(* Logix 5000 project; controller cow Emulate 5570 rev 36.11; software revision 36.00; part 3 of 6 *)

VAR_GLOBAL   (* controller tags *)
   B111 : MotorX := (InterLock := 1, SP := 1, LSK := 1);
   B113 : MotorX := (LSK := 1);
   B116 : MotorX := (LSK := 1);
   B126 : MotorX := (InterLock := 1, SP := 1, LSK := 1, CLEAN := 1);
   B160 : MotorX := (LSK := 1);
   B280 : Divider := (LS3 := 1, LS_ON := 1, Simulate := 3);
   B3 : INT[50] := ([0] := 1, [2] := 896, [3] := 15824, [6] := 24508, [7] := 19455, [8] := 677, [16] := 7, [18] := 1503, [22] := 4736, [23] := 160, [24] := 2145, [26] := -22782, [28] := -22484, [29] := 21, [30] := 768, [33] := 11328, [34] := 24701, [35] := 12288, [40] := 4, [41] := 4, [42] := 816, [43] := -19680, [44] := -21846, [45] := -32054, [46] := 194, [47] := 26775);
   B353 : Gate := (LSK := 1);
   B354 : Gate := (LSK := 1);
   B361 : Branch_SV2 := (LSX := 1, GLX := 1);
   B362 : Branch_SV2 := (LSY := 1, GLY := 1);
   B363 : Branch_SV2 := (LSY := 1, GLY := 1);
   B364 : Branch_SV2 := (LSY := 1, GLY := 1);
   B365 : Branch_SV2 := (LSX := 1, GLX := 1);
   B367 : Branch_SV2 := (LSX := 1, GLX := 1);
   B410 : MotorX := (LSK := 1);
   B420 : MotorX := (LSK := 1);
   Bin01 : ALIAS FOR rcp_Big_Bin[0];
   Bin02 : ALIAS FOR rcp_Big_Bin[1];
   Bin03 : ALIAS FOR rcp_Big_Bin[2];
   Bin04 : ALIAS FOR rcp_Big_Bin[3];
   Bin05 : ALIAS FOR rcp_Big_Bin[4];
   Bin06 : ALIAS FOR rcp_Big_Bin[5];
   Bin07 : ALIAS FOR rcp_Big_Bin[6];
   Bin08 : ALIAS FOR rcp_Big_Bin[7];
   Bin09 : ALIAS FOR rcp_Big_Bin[8];
   Bin10 : ALIAS FOR rcp_Big_Bin[9];
   Bin11 : ALIAS FOR rcp_Big_Bin[10];
   Bin12 : ALIAS FOR rcp_Big_Bin[11];
   Bin13 : ALIAS FOR rcp_Big_Bin[12];
   Bin14 : ALIAS FOR rcp_Big_Bin[13];
   Bin15 : ALIAS FOR rcp_Big_Bin[14];
   Bin16 : ALIAS FOR rcp_Big_Bin[15];
   Buf_LenSent : DINT := 8;
   D121 : MotorX := (LSK := 1);
   D162 : MotorX := (LSK := 1);
   D163 : MotorX := (LSK := 1);
   D164 : MotorX := (LSK := 1);
   D230 : MotorX := (LSK := 1);
   D361 : Branch_SV2 := (LSY := 1, GLY := 1);
   D380 : MotorX := (LSK := 1);
   D411 : MotorX := (LSK := 1);
   D421 : MotorX := (LSK := 1);
   DateTimes : STRING := '2026/06/05  08:19:56';
   Delete_All_MSG : MESSAGE;
        MessageParameters(ServiceCode := 16#0051, ...)
   E112 : MotorX := (LL := 1, Auto := 1, LSK := 1);   // B112
   E112_Have : BOOL;
   E112_Have_Flash : BOOL;
   E120 : MotorX := (Auto := 1, SP := 1, LSK := 1, CLEAN := 1);   // B120
   E141 : MotorX := (Auto := 1, SP := 1, LSK := 1);   // B141
   E142 : MotorX := (Auto := 1, SP := 1, LSK := 1);
   E143 : MotorX := (Auto := 1, LSK := 1);
   E144 : MotorX := (Auto := 1, LSK := 1);
   E145 : MotorX := (Auto := 1, SP := 1, LSK := 1);
   E146 : MotorX := (Auto := 1, LSK := 1);
   E147 : MotorX := (Auto := 1, LSK := 1);
   E148 : MotorX := (Auto := 1, LSK := 1);
   E149 : MotorX := (Auto := 1, LSK := 1);
   E14A : MotorX := (Auto := 1, LSK := 1);
   E14B : MotorX := (Auto := 1, LSK := 1);
   E14C : MotorX := (Auto := 1, LSK := 1);
   E14D : MotorX := (Auto := 1, LSK := 1);
   E14E : MotorX := (Auto := 1, LSK := 1);
   E14F : MotorX := (Auto := 1, LSK := 1);
   E14G : MotorX := (Auto := 1, LSK := 1);
   E331 : SCALE_WEIGHT;
   E340 : Valve := (LSK := 1, Auto := 1, PB := 1);
   E351 : Valve := (LSK := 1, Auto := 1);
   E352 : Valve := (LSK := 1, Auto := 1);
   E45A : Air_Hammer := (MotorType := 1);
   E45B : Air_Hammer;
   E45C : Air_Hammer;
   EINV : Inverter := (Manual_HZ := 10);
   F090 : MotorX := (LSK := 1);
   F124 : MotorX := (LSK := 1);
   F125 : MotorX := (LSK := 1);
   F140 : MotorX := (LSK := 1);
   F167 : MotorX := (LSK := 1);
   F168 : MotorX := (LSK := 1);
   F240 : MotorX := (LSK := 1);
   F270 : MotorX := (LSK := 1);
   F363 : Branch_SV2 := (LSY := 1, GLY := 1);
   F364 : Branch_SV2 := (LSY := 1, GLY := 1);
   F413 : MotorX := (LSK := 1);
   F441 : MotorX := (LSK := 1);
   F560 : MotorX := (LSK := 1);
   F561 : MotorX := (LSK := 1);
   LED0_Create_Sock_MSG : MESSAGE;
        MessageParameters(ServiceCode := 16#004b, LocalElement := LED_SOCKET[0], DestinationTag := LED_Instance[0], ...)
   LED0_Write_Data_MSG : MESSAGE;
        MessageParameters(ServiceCode := 16#004e, LocalElement := LED_Write_Data_Out[0], DestinationTag := Buf_LenSent, ...)
   LED_Batch_seq : DINT := 1;
   LED_Batch_Total : ALIAS FOR rcp_Recipe.BatchSet;
   Led_Hand_PartNumber : DINT;
   Led_Hand_RealWeight : REAL;
   LED_Hand_SetWeight : REAL;
   LED_Instance : DINT[16] := ([0] := 18562, [1] := 31683, [2] := 27332, [3] := 24000, [4] := 22593, [5] := 19589, [6] := 24710, [7] := 29255, [8] := 16968);
   LED_SOCKET : REQUEST_PARAMETERS[16] := ([0].Type := 2, [0].Addr.Family := 2, [0].Addr.Port := 123, [1].Type := 2, [1].Addr.Family := 2, [1].Addr.Port := 121, [2].Type := 2, [2].Addr.Family := 2, [2].Addr.Port := 221, [3].Type := 2, [3].Addr.Family := 2, [3].Addr.Port := 122, [4].Type := 2, [4].Addr.Family := 2, [4].Addr.Port := 222, [5].Type := 2, [5].Addr.Family := 2, [5].Addr.Port := 223, [6].Type := 2, [6].Addr.Family := 2, [6].Addr.Port := 124, [7].Type := 2, [7].Addr.Family := 2, [7].Addr.Port := 125, [8].Type := 2, [8].Addr.Family := 2, [8].Addr.Port := 226);
   Led_string : STRING[16] := ([0] := 'Test$00$00$00$00$00$00 2-1      ', [1] := '2026/04/29  10:28:13', [2] := '730000600  100.0 Kg ', [3] := 'BIN:41 3016E 5.00 t ', [4] := 'BIN:34 2410$00$00- 6.00t', [5] := '2026/04/29  10:28:13', [6] := 'S19-B8-2001B$00-99.0t ', [7] := 'S0-B139-3015$00$00- 3.0t', [8] := 'BIN1 2001F$00-30.00t  ');
   LED_Write_Data_Out : WRT_DATA[16] := ([0].Timeout := 20000, [0].ToAddr.Family := 2, [0].ToAddr.Port := 8001, [0].ToAddr.Addr := 16#c101_017b, [0].Buffer.LEN := 31, [0].Buffer.BUFF[0] := 2, [0].Buffer.BUFF[1] := 90, [0].Buffer.BUFF[2] := 48, [0].Buffer.BUFF[3] := -95, [0].Buffer.BUFF[4] := 1, [0].Buffer.BUFF[5] := 1, [0].Buffer.BUFF[6] := 78, [0].Buffer.BUFF[7] := -48, [0].Buffer.BUFF[8] := 55, [0].Buffer.BUFF[9] := 55, [0].Buffer.BUFF[10] := 48, [0].Buffer.BUFF[11] := 48, [0].Buffer.BUFF[12] := 51, [0].Buffer.BUFF[13] := 49, [0].Buffer.BUFF[14] := 51, [0].Buffer.BUFF[15] := 57, [0].Buffer.BUFF[16] := 48, [0].Buffer.BUFF[17] := 100, [0].Buffer.BUFF[18] := 32, [0].Buffer.BUFF[19] := 53, [0].Buffer.BUFF[20] := 45, [0].Buffer.BUFF[21] := 51, [0].Buffer.BUFF[22] := 32, [0].Buffer.BUFF[23] := 32, [0].Buffer.BUFF[24] := 32, [0].Buffer.BUFF[25] := 32, [0].Buffer.BUFF[26] := 32, [0].Buffer.BUFF[27] := 32, [0].Buffer.BUFF[28] := 82, [0].Buffer.BUFF[29] := 80, [0].Buffer.BUFF[30] := 3, [0].Buffer.BUFF[31] := 46, [0].Buffer.BUFF[32] := 48, [0].Buffer.BUFF[33] := 82, [0].Buffer.BUFF[34] := 51, [0].Buffer.BUFF[35] := 3, [0].Buffer.BUFF[84] := 31, [0].Buffer.BUFF[88] := 2, [0].Buffer.BUFF[89] := 90, [0].Buffer.BUFF[90] := 48, [0].Buffer.BUFF[91] := -95, [0].Buffer.BUFF[92] := 1, [0].Buffer.BUFF[93] := 1, [0].Buffer.BUFF[94] := 78, [0].Buffer.BUFF[95] := -48, [0].Buffer.BUFF[96] := 50, [0].Buffer.BUFF[97] := 48, [0].Buffer.BUFF[98] := 50, [0].Buffer.BUFF[99] := 54, [0].Buffer.BUFF[100] := 47, [0].Buffer.BUFF[101] := 48, [0].Buffer.BUFF[102] := 52, [0].Buffer.BUFF[103] := 47, [0].Buffer.BUFF[104] := 50, [0].Buffer.BUFF[105] := 57,
        [0].Buffer.BUFF[106] := 32, [0].Buffer.BUFF[107] := 32, [0].Buffer.BUFF[108] := 49, [0].Buffer.BUFF[109] := 48, [0].Buffer.BUFF[110] := 58, [0].Buffer.BUFF[111] := 50, [0].Buffer.BUFF[112] := 56, [0].Buffer.BUFF[113] := 58, [0].Buffer.BUFF[114] := 48, [0].Buffer.BUFF[115] := 56, [0].Buffer.BUFF[116] := 82, [0].Buffer.BUFF[117] := 13, [0].Buffer.BUFF[118] := 3, [0].Buffer.BUFF[172] := 31, [0].Buffer.BUFF[176] := 2, [0].Buffer.BUFF[177] := 90, [0].Buffer.BUFF[178] := 48, [0].Buffer.BUFF[179] := -95, [0].Buffer.BUFF[180] := 1, [0].Buffer.BUFF[181] := 1, [0].Buffer.BUFF[182] := 78, [0].Buffer.BUFF[183] := -48, [0].Buffer.BUFF[184] := 55, [0].Buffer.BUFF[185] := 51, [0].Buffer.BUFF[186] := 48, [0].Buffer.BUFF[187] := 48, [0].Buffer.BUFF[188] := 48, [0].Buffer.BUFF[189] := 48, [0].Buffer.BUFF[190] := 54, [0].Buffer.BUFF[191] := 48, [0].Buffer.BUFF[192] := 48, [0].Buffer.BUFF[193] := 32, [0].Buffer.BUFF[194] := 32, [0].Buffer.BUFF[195] := 49, [0].Buffer.BUFF[196] := 48, [0].Buffer.BUFF[197] := 48, [0].Buffer.BUFF[198] := 46, [0].Buffer.BUFF[199] := 48, [0].Buffer.BUFF[200] := 32, [0].Buffer.BUFF[201] := 75, [0].Buffer.BUFF[202] := 103, [0].Buffer.BUFF[203] := 32, [0].Buffer.BUFF[204] := 82, [0].Buffer.BUFF[205] := 54, [0].Buffer.BUFF[206] := 3, [0].Buffer.BUFF[260] := 31, [0].Buffer.BUFF[264] := 2, [0].Buffer.BUFF[265] := 90, [0].Buffer.BUFF[266] := 48, [0].Buffer.BUFF[267] := -95, [0].Buffer.BUFF[268] := 1, [0].Buffer.BUFF[269] := 1, [0].Buffer.BUFF[270] := 78, [0].Buffer.BUFF[271] := -48, [0].Buffer.BUFF[272] := 66, [0].Buffer.BUFF[273] := 73, [0].Buffer.BUFF[274] := 78, [0].Buffer.BUFF[275] := 58, [0].Buffer.BUFF[276] := 52, [0].Buffer.BUFF[277] := 49,
        [0].Buffer.BUFF[278] := 32, [0].Buffer.BUFF[279] := 51, [0].Buffer.BUFF[280] := 48, [0].Buffer.BUFF[281] := 49, [0].Buffer.BUFF[282] := 54, [0].Buffer.BUFF[283] := 69, [0].Buffer.BUFF[284] := 32, [0].Buffer.BUFF[285] := 53, [0].Buffer.BUFF[286] := 46, [0].Buffer.BUFF[287] := 48, [0].Buffer.BUFF[288] := 48, [0].Buffer.BUFF[289] := 32, [0].Buffer.BUFF[290] := 116, [0].Buffer.BUFF[291] := 32, [0].Buffer.BUFF[292] := 82, [0].Buffer.BUFF[293] := 83, [0].Buffer.BUFF[294] := 3, [0].Buffer.BUFF[348] := 31, [0].Buffer.BUFF[352] := 2, [0].Buffer.BUFF[353] := 90, [0].Buffer.BUFF[354] := 48, [0].Buffer.BUFF[355] := -95, [0].Buffer.BUFF[356] := 1, [0].Buffer.BUFF[357] := 1, [0].Buffer.BUFF[358] := 78, [0].Buffer.BUFF[359] := -48, [0].Buffer.BUFF[360] := 66, [0].Buffer.BUFF[361] := 73, [0].Buffer.BUFF[362] := 78, [0].Buffer.BUFF[363] := 58, [0].Buffer.BUFF[364] := 51, [0].Buffer.BUFF[365] := 52, [0].Buffer.BUFF[366] := 32, [0].Buffer.BUFF[367] := 50, [0].Buffer.BUFF[368] := 52, [0].Buffer.BUFF[369] := 49, [0].Buffer.BUFF[370] := 48, [0].Buffer.BUFF[373] := 45, [0].Buffer.BUFF[374] := 32, [0].Buffer.BUFF[375] := 54, [0].Buffer.BUFF[376] := 46, [0].Buffer.BUFF[377] := 48, [0].Buffer.BUFF[378] := 48, [0].Buffer.BUFF[379] := 116, [0].Buffer.BUFF[380] := 82, [0].Buffer.BUFF[381] := 57, [0].Buffer.BUFF[382] := 3, [0].Buffer.BUFF[436] := 31, [0].Buffer.BUFF[440] := 2, [0].Buffer.BUFF[441] := 90, [0].Buffer.BUFF[442] := 48, [0].Buffer.BUFF[443] := -95, [0].Buffer.BUFF[444] := 1, [0].Buffer.BUFF[445] := 1, [0].Buffer.BUFF[446] := 78, [0].Buffer.BUFF[447] := -48, [0].Buffer.BUFF[448] := 50, [0].Buffer.BUFF[449] := 48, [0].Buffer.BUFF[450] := 50, [0].Buffer.BUFF[451] := 54,
        [0].Buffer.BUFF[452] := 47, [0].Buffer.BUFF[453] := 48, [0].Buffer.BUFF[454] := 52, [0].Buffer.BUFF[455] := 47, [0].Buffer.BUFF[456] := 50, [0].Buffer.BUFF[457] := 57, [0].Buffer.BUFF[458] := 32, [0].Buffer.BUFF[459] := 32, [0].Buffer.BUFF[460] := 49, [0].Buffer.BUFF[461] := 48, [0].Buffer.BUFF[462] := 58, [0].Buffer.BUFF[463] := 50, [0].Buffer.BUFF[464] := 56, [0].Buffer.BUFF[465] := 58, [0].Buffer.BUFF[466] := 48, [0].Buffer.BUFF[467] := 56, [0].Buffer.BUFF[468] := 82, [0].Buffer.BUFF[469] := 13, [0].Buffer.BUFF[470] := 3, [1].ToAddr.Family := 2, [1].ToAddr.Port := 8001, [1].ToAddr.Addr := 16#c101_0179, [1].Buffer.LEN := 31, [1].Buffer.BUFF[0] := 2, [1].Buffer.BUFF[1] := 90, [1].Buffer.BUFF[2] := 48, [1].Buffer.BUFF[3] := -95, [1].Buffer.BUFF[4] := 1, [1].Buffer.BUFF[5] := 1, [1].Buffer.BUFF[6] := 78, [1].Buffer.BUFF[7] := -48, [1].Buffer.BUFF[8] := 50, [1].Buffer.BUFF[9] := 48, [1].Buffer.BUFF[10] := 50, [1].Buffer.BUFF[11] := 54, [1].Buffer.BUFF[12] := 47, [1].Buffer.BUFF[13] := 48, [1].Buffer.BUFF[14] := 52, [1].Buffer.BUFF[15] := 47, [1].Buffer.BUFF[16] := 50, [1].Buffer.BUFF[17] := 57, [1].Buffer.BUFF[18] := 32, [1].Buffer.BUFF[19] := 32, [1].Buffer.BUFF[20] := 49, [1].Buffer.BUFF[21] := 48, [1].Buffer.BUFF[22] := 58, [1].Buffer.BUFF[23] := 50, [1].Buffer.BUFF[24] := 56, [1].Buffer.BUFF[25] := 58, [1].Buffer.BUFF[26] := 48, [1].Buffer.BUFF[27] := 55, [1].Buffer.BUFF[28] := 82, [1].Buffer.BUFF[29] := 2, [1].Buffer.BUFF[30] := 3, [1].Buffer.BUFF[84] := 31, [1].Buffer.BUFF[88] := 2, [1].Buffer.BUFF[89] := 90, [1].Buffer.BUFF[90] := 48, [1].Buffer.BUFF[91] := -95, [1].Buffer.BUFF[92] := 1,
        [1].Buffer.BUFF[93] := 1, [1].Buffer.BUFF[94] := 78, [1].Buffer.BUFF[95] := -48, [1].Buffer.BUFF[96] := 55, [1].Buffer.BUFF[97] := 51, [1].Buffer.BUFF[98] := 48, [1].Buffer.BUFF[99] := 48, [1].Buffer.BUFF[100] := 48, [1].Buffer.BUFF[101] := 48, [1].Buffer.BUFF[102] := 54, [1].Buffer.BUFF[103] := 48, [1].Buffer.BUFF[104] := 48, [1].Buffer.BUFF[105] := 32, [1].Buffer.BUFF[106] := 32, [1].Buffer.BUFF[107] := 49, [1].Buffer.BUFF[108] := 48, [1].Buffer.BUFF[109] := 48, [1].Buffer.BUFF[110] := 46, [1].Buffer.BUFF[111] := 48, [1].Buffer.BUFF[112] := 32, [1].Buffer.BUFF[113] := 75, [1].Buffer.BUFF[114] := 103, [1].Buffer.BUFF[115] := 32, [1].Buffer.BUFF[116] := 82, [1].Buffer.BUFF[117] := 54, [1].Buffer.BUFF[118] := 3, [1].Buffer.BUFF[172] := 31, [1].Buffer.BUFF[176] := 2, [1].Buffer.BUFF[177] := 90, [1].Buffer.BUFF[178] := 48, [1].Buffer.BUFF[179] := -95, [1].Buffer.BUFF[180] := 1, [1].Buffer.BUFF[181] := 1, [1].Buffer.BUFF[182] := 78, [1].Buffer.BUFF[183] := -48, [1].Buffer.BUFF[184] := 66, [1].Buffer.BUFF[185] := 73, [1].Buffer.BUFF[186] := 78, [1].Buffer.BUFF[187] := 58, [1].Buffer.BUFF[188] := 52, [1].Buffer.BUFF[189] := 49, [1].Buffer.BUFF[190] := 32, [1].Buffer.BUFF[191] := 51, [1].Buffer.BUFF[192] := 48, [1].Buffer.BUFF[193] := 49, [1].Buffer.BUFF[194] := 54, [1].Buffer.BUFF[195] := 69, [1].Buffer.BUFF[196] := 32, [1].Buffer.BUFF[197] := 53, [1].Buffer.BUFF[198] := 46, [1].Buffer.BUFF[199] := 48, [1].Buffer.BUFF[200] := 48, [1].Buffer.BUFF[201] := 32, [1].Buffer.BUFF[202] := 116, [1].Buffer.BUFF[203] := 32, [1].Buffer.BUFF[204] := 82, [1].Buffer.BUFF[205] := 83, [1].Buffer.BUFF[206] := 3, [1].Buffer.BUFF[260] := 31, [1].Buffer.BUFF[264] := 2,
        [1].Buffer.BUFF[265] := 90, [1].Buffer.BUFF[266] := 48, [1].Buffer.BUFF[267] := -95, [1].Buffer.BUFF[268] := 1, [1].Buffer.BUFF[269] := 1, [1].Buffer.BUFF[270] := 78, [1].Buffer.BUFF[271] := -48, [1].Buffer.BUFF[272] := 66, [1].Buffer.BUFF[273] := 73, [1].Buffer.BUFF[274] := 78, [1].Buffer.BUFF[275] := 58, [1].Buffer.BUFF[276] := 51, [1].Buffer.BUFF[277] := 52, [1].Buffer.BUFF[278] := 32, [1].Buffer.BUFF[279] := 50, [1].Buffer.BUFF[280] := 52, [1].Buffer.BUFF[281] := 49, [1].Buffer.BUFF[282] := 48, [1].Buffer.BUFF[285] := 45, [1].Buffer.BUFF[286] := 32, [1].Buffer.BUFF[287] := 54, [1].Buffer.BUFF[288] := 46, [1].Buffer.BUFF[289] := 48, [1].Buffer.BUFF[290] := 48, [1].Buffer.BUFF[291] := 116, [1].Buffer.BUFF[292] := 82, [1].Buffer.BUFF[293] := 57, [1].Buffer.BUFF[294] := 3, [1].Buffer.BUFF[348] := 31, [1].Buffer.BUFF[352] := 2, [1].Buffer.BUFF[353] := 90, [1].Buffer.BUFF[354] := 48, [1].Buffer.BUFF[355] := -95, [1].Buffer.BUFF[356] := 1, [1].Buffer.BUFF[357] := 1, [1].Buffer.BUFF[358] := 78, [1].Buffer.BUFF[359] := -48, [1].Buffer.BUFF[360] := 50, [1].Buffer.BUFF[361] := 48, [1].Buffer.BUFF[362] := 50, [1].Buffer.BUFF[363] := 54, [1].Buffer.BUFF[364] := 47, [1].Buffer.BUFF[365] := 48, [1].Buffer.BUFF[366] := 52, [1].Buffer.BUFF[367] := 47, [1].Buffer.BUFF[368] := 50, [1].Buffer.BUFF[369] := 57, [1].Buffer.BUFF[370] := 32, [1].Buffer.BUFF[371] := 32, [1].Buffer.BUFF[372] := 49, [1].Buffer.BUFF[373] := 48, [1].Buffer.BUFF[374] := 58, [1].Buffer.BUFF[375] := 50, [1].Buffer.BUFF[376] := 56, [1].Buffer.BUFF[377] := 58, [1].Buffer.BUFF[378] := 48, [1].Buffer.BUFF[379] := 55, [1].Buffer.BUFF[380] := 82, [1].Buffer.BUFF[381] := 2, [1].Buffer.BUFF[382] := 3,
        [1].Buffer.BUFF[436] := 31, [1].Buffer.BUFF[440] := 2, [1].Buffer.BUFF[441] := 90, [1].Buffer.BUFF[442] := 48, [1].Buffer.BUFF[443] := -95, [1].Buffer.BUFF[444] := 1, [1].Buffer.BUFF[445] := 1, [1].Buffer.BUFF[446] := 78, [1].Buffer.BUFF[447] := -48, [1].Buffer.BUFF[448] := 83, [1].Buffer.BUFF[449] := 49, [1].Buffer.BUFF[450] := 57, [1].Buffer.BUFF[451] := 45, [1].Buffer.BUFF[452] := 66, [1].Buffer.BUFF[453] := 56, [1].Buffer.BUFF[454] := 45, [1].Buffer.BUFF[455] := 50, [1].Buffer.BUFF[456] := 48, [1].Buffer.BUFF[457] := 48, [1].Buffer.BUFF[458] := 49, [1].Buffer.BUFF[459] := 66, [1].Buffer.BUFF[461] := 45, [1].Buffer.BUFF[462] := 57, [1].Buffer.BUFF[463] := 57, [1].Buffer.BUFF[464] := 46, [1].Buffer.BUFF[465] := 48, [1].Buffer.BUFF[466] := 116, [1].Buffer.BUFF[467] := 32, [1].Buffer.BUFF[468] := 82, [1].Buffer.BUFF[470] := 3, [2].ToAddr.Family := 2, [2].ToAddr.Port := 8002, [2].ToAddr.Addr := 16#c101_0179, [2].Buffer.LEN := 31, [2].Buffer.BUFF[0] := 2, [2].Buffer.BUFF[1] := 90, [2].Buffer.BUFF[2] := 48, [2].Buffer.BUFF[3] := -95, [2].Buffer.BUFF[4] := 1, [2].Buffer.BUFF[5] := 1, [2].Buffer.BUFF[6] := 78, [2].Buffer.BUFF[7] := -48, [2].Buffer.BUFF[8] := 55, [2].Buffer.BUFF[9] := 51, [2].Buffer.BUFF[10] := 48, [2].Buffer.BUFF[11] := 48, [2].Buffer.BUFF[12] := 48, [2].Buffer.BUFF[13] := 48, [2].Buffer.BUFF[14] := 54, [2].Buffer.BUFF[15] := 48, [2].Buffer.BUFF[16] := 48, [2].Buffer.BUFF[17] := 32, [2].Buffer.BUFF[18] := 32, [2].Buffer.BUFF[19] := 49, [2].Buffer.BUFF[20] := 48, [2].Buffer.BUFF[21] := 48, [2].Buffer.BUFF[22] := 46, [2].Buffer.BUFF[23] := 48, [2].Buffer.BUFF[24] := 32, [2].Buffer.BUFF[25] := 75,
        [2].Buffer.BUFF[26] := 103, [2].Buffer.BUFF[27] := 32, [2].Buffer.BUFF[28] := 82, [2].Buffer.BUFF[29] := 54, [2].Buffer.BUFF[30] := 3, [2].Buffer.BUFF[84] := 31, [2].Buffer.BUFF[88] := 2, [2].Buffer.BUFF[89] := 90, [2].Buffer.BUFF[90] := 48, [2].Buffer.BUFF[91] := -95, [2].Buffer.BUFF[92] := 1, [2].Buffer.BUFF[93] := 1, [2].Buffer.BUFF[94] := 78, [2].Buffer.BUFF[95] := -48, [2].Buffer.BUFF[96] := 66, [2].Buffer.BUFF[97] := 73, [2].Buffer.BUFF[98] := 78, [2].Buffer.BUFF[99] := 58, [2].Buffer.BUFF[100] := 52, [2].Buffer.BUFF[101] := 49, [2].Buffer.BUFF[102] := 32, [2].Buffer.BUFF[103] := 51, [2].Buffer.BUFF[104] := 48, [2].Buffer.BUFF[105] := 49, [2].Buffer.BUFF[106] := 54, [2].Buffer.BUFF[107] := 69, [2].Buffer.BUFF[108] := 32, [2].Buffer.BUFF[109] := 53, [2].Buffer.BUFF[110] := 46, [2].Buffer.BUFF[111] := 48, [2].Buffer.BUFF[112] := 48, [2].Buffer.BUFF[113] := 32, [2].Buffer.BUFF[114] := 116, [2].Buffer.BUFF[115] := 32, [2].Buffer.BUFF[116] := 82, [2].Buffer.BUFF[117] := 83, [2].Buffer.BUFF[118] := 3, [2].Buffer.BUFF[172] := 31, [2].Buffer.BUFF[176] := 2, [2].Buffer.BUFF[177] := 90, [2].Buffer.BUFF[178] := 48, [2].Buffer.BUFF[179] := -95, [2].Buffer.BUFF[180] := 1, [2].Buffer.BUFF[181] := 1, [2].Buffer.BUFF[182] := 78, [2].Buffer.BUFF[183] := -48, [2].Buffer.BUFF[184] := 66, [2].Buffer.BUFF[185] := 73, [2].Buffer.BUFF[186] := 78, [2].Buffer.BUFF[187] := 58, [2].Buffer.BUFF[188] := 51, [2].Buffer.BUFF[189] := 52, [2].Buffer.BUFF[190] := 32, [2].Buffer.BUFF[191] := 50, [2].Buffer.BUFF[192] := 52, [2].Buffer.BUFF[193] := 49, [2].Buffer.BUFF[194] := 48, [2].Buffer.BUFF[197] := 45, [2].Buffer.BUFF[198] := 32, [2].Buffer.BUFF[199] := 54,
        [2].Buffer.BUFF[200] := 46, [2].Buffer.BUFF[201] := 48, [2].Buffer.BUFF[202] := 48, [2].Buffer.BUFF[203] := 116, [2].Buffer.BUFF[204] := 82, [2].Buffer.BUFF[205] := 57, [2].Buffer.BUFF[206] := 3, [2].Buffer.BUFF[260] := 31, [2].Buffer.BUFF[264] := 2, [2].Buffer.BUFF[265] := 90, [2].Buffer.BUFF[266] := 48, [2].Buffer.BUFF[267] := -95, [2].Buffer.BUFF[268] := 1, [2].Buffer.BUFF[269] := 1, [2].Buffer.BUFF[270] := 78, [2].Buffer.BUFF[271] := -48, [2].Buffer.BUFF[272] := 50, [2].Buffer.BUFF[273] := 48, [2].Buffer.BUFF[274] := 50, [2].Buffer.BUFF[275] := 54, [2].Buffer.BUFF[276] := 47, [2].Buffer.BUFF[277] := 48, [2].Buffer.BUFF[278] := 52, [2].Buffer.BUFF[279] := 47, [2].Buffer.BUFF[280] := 50, [2].Buffer.BUFF[281] := 57, [2].Buffer.BUFF[282] := 32, [2].Buffer.BUFF[283] := 32, [2].Buffer.BUFF[284] := 49, [2].Buffer.BUFF[285] := 48, [2].Buffer.BUFF[286] := 58, [2].Buffer.BUFF[287] := 50, [2].Buffer.BUFF[288] := 56, [2].Buffer.BUFF[289] := 58, [2].Buffer.BUFF[290] := 48, [2].Buffer.BUFF[291] := 55, [2].Buffer.BUFF[292] := 82, [2].Buffer.BUFF[293] := 2, [2].Buffer.BUFF[294] := 3, [2].Buffer.BUFF[348] := 31, [2].Buffer.BUFF[352] := 2, [2].Buffer.BUFF[353] := 90, [2].Buffer.BUFF[354] := 48, [2].Buffer.BUFF[355] := -95, [2].Buffer.BUFF[356] := 1, [2].Buffer.BUFF[357] := 1, [2].Buffer.BUFF[358] := 78, [2].Buffer.BUFF[359] := -48, [2].Buffer.BUFF[360] := 83, [2].Buffer.BUFF[361] := 49, [2].Buffer.BUFF[362] := 57, [2].Buffer.BUFF[363] := 45, [2].Buffer.BUFF[364] := 66, [2].Buffer.BUFF[365] := 56, [2].Buffer.BUFF[366] := 45, [2].Buffer.BUFF[367] := 50, [2].Buffer.BUFF[368] := 48, [2].Buffer.BUFF[369] := 48, [2].Buffer.BUFF[370] := 49, [2].Buffer.BUFF[371] := 66,
        [2].Buffer.BUFF[373] := 45, [2].Buffer.BUFF[374] := 57, [2].Buffer.BUFF[375] := 57, [2].Buffer.BUFF[376] := 46, [2].Buffer.BUFF[377] := 48, [2].Buffer.BUFF[378] := 116, [2].Buffer.BUFF[379] := 32, [2].Buffer.BUFF[380] := 82, [2].Buffer.BUFF[382] := 3, [2].Buffer.BUFF[436] := 31, [2].Buffer.BUFF[440] := 2, [2].Buffer.BUFF[441] := 90, [2].Buffer.BUFF[442] := 48, [2].Buffer.BUFF[443] := -95, [2].Buffer.BUFF[444] := 1, [2].Buffer.BUFF[445] := 1, [2].Buffer.BUFF[446] := 78, [2].Buffer.BUFF[447] := -48, [2].Buffer.BUFF[448] := 83, [2].Buffer.BUFF[449] := 48, [2].Buffer.BUFF[450] := 45, [2].Buffer.BUFF[451] := 66, [2].Buffer.BUFF[452] := 49, [2].Buffer.BUFF[453] := 51, [2].Buffer.BUFF[454] := 57, [2].Buffer.BUFF[455] := 45, [2].Buffer.BUFF[456] := 51, [2].Buffer.BUFF[457] := 48, [2].Buffer.BUFF[458] := 49, [2].Buffer.BUFF[459] := 53, [2].Buffer.BUFF[462] := 45, [2].Buffer.BUFF[463] := 32, [2].Buffer.BUFF[464] := 51, [2].Buffer.BUFF[465] := 46, [2].Buffer.BUFF[466] := 48, [2].Buffer.BUFF[467] := 116, [2].Buffer.BUFF[468] := 82, [2].Buffer.BUFF[469] := 78, [2].Buffer.BUFF[470] := 3, [3].ToAddr.Family := 2, [3].ToAddr.Port := 8001, [3].ToAddr.Addr := 16#c101_017a, [3].Buffer.LEN := 31, [3].Buffer.BUFF[0] := 2, [3].Buffer.BUFF[1] := 90, [3].Buffer.BUFF[2] := 48, [3].Buffer.BUFF[3] := -95, [3].Buffer.BUFF[4] := 1, [3].Buffer.BUFF[5] := 1, [3].Buffer.BUFF[6] := 78, [3].Buffer.BUFF[7] := -48, [3].Buffer.BUFF[8] := 66, [3].Buffer.BUFF[9] := 73, [3].Buffer.BUFF[10] := 78, [3].Buffer.BUFF[11] := 58, [3].Buffer.BUFF[12] := 52, [3].Buffer.BUFF[13] := 49, [3].Buffer.BUFF[14] := 32, [3].Buffer.BUFF[15] := 51, [3].Buffer.BUFF[16] := 48,
        [3].Buffer.BUFF[17] := 49, [3].Buffer.BUFF[18] := 54, [3].Buffer.BUFF[19] := 69, [3].Buffer.BUFF[20] := 32, [3].Buffer.BUFF[21] := 53, [3].Buffer.BUFF[22] := 46, [3].Buffer.BUFF[23] := 48, [3].Buffer.BUFF[24] := 48, [3].Buffer.BUFF[25] := 32, [3].Buffer.BUFF[26] := 116, [3].Buffer.BUFF[27] := 32, [3].Buffer.BUFF[28] := 82, [3].Buffer.BUFF[29] := 83, [3].Buffer.BUFF[30] := 3, [3].Buffer.BUFF[84] := 31, [3].Buffer.BUFF[88] := 2, [3].Buffer.BUFF[89] := 90, [3].Buffer.BUFF[90] := 48, [3].Buffer.BUFF[91] := -95, [3].Buffer.BUFF[92] := 1, [3].Buffer.BUFF[93] := 1, [3].Buffer.BUFF[94] := 78, [3].Buffer.BUFF[95] := -48, [3].Buffer.BUFF[96] := 66, [3].Buffer.BUFF[97] := 73, [3].Buffer.BUFF[98] := 78, [3].Buffer.BUFF[99] := 58, [3].Buffer.BUFF[100] := 51, [3].Buffer.BUFF[101] := 52, [3].Buffer.BUFF[102] := 32, [3].Buffer.BUFF[103] := 50, [3].Buffer.BUFF[104] := 52, [3].Buffer.BUFF[105] := 49, [3].Buffer.BUFF[106] := 48, [3].Buffer.BUFF[109] := 45, [3].Buffer.BUFF[110] := 32, [3].Buffer.BUFF[111] := 54, [3].Buffer.BUFF[112] := 46, [3].Buffer.BUFF[113] := 48, [3].Buffer.BUFF[114] := 48, [3].Buffer.BUFF[115] := 116, [3].Buffer.BUFF[116] := 82, [3].Buffer.BUFF[117] := 57, [3].Buffer.BUFF[118] := 3, [3].Buffer.BUFF[172] := 31, [3].Buffer.BUFF[176] := 2, [3].Buffer.BUFF[177] := 90, [3].Buffer.BUFF[178] := 48, [3].Buffer.BUFF[179] := -95, [3].Buffer.BUFF[180] := 1, [3].Buffer.BUFF[181] := 1, [3].Buffer.BUFF[182] := 78, [3].Buffer.BUFF[183] := -48, [3].Buffer.BUFF[184] := 50, [3].Buffer.BUFF[185] := 48, [3].Buffer.BUFF[186] := 50, [3].Buffer.BUFF[187] := 54, [3].Buffer.BUFF[188] := 47, [3].Buffer.BUFF[189] := 48, [3].Buffer.BUFF[190] := 52,
        [3].Buffer.BUFF[191] := 47, [3].Buffer.BUFF[192] := 50, [3].Buffer.BUFF[193] := 57, [3].Buffer.BUFF[194] := 32, [3].Buffer.BUFF[195] := 32, [3].Buffer.BUFF[196] := 49, [3].Buffer.BUFF[197] := 48, [3].Buffer.BUFF[198] := 58, [3].Buffer.BUFF[199] := 50, [3].Buffer.BUFF[200] := 56, [3].Buffer.BUFF[201] := 58, [3].Buffer.BUFF[202] := 48, [3].Buffer.BUFF[203] := 55, [3].Buffer.BUFF[204] := 82, [3].Buffer.BUFF[205] := 2, [3].Buffer.BUFF[206] := 3, [3].Buffer.BUFF[260] := 31, [3].Buffer.BUFF[264] := 2, [3].Buffer.BUFF[265] := 90, [3].Buffer.BUFF[266] := 48, [3].Buffer.BUFF[267] := -95, [3].Buffer.BUFF[268] := 1, [3].Buffer.BUFF[269] := 1, [3].Buffer.BUFF[270] := 78, [3].Buffer.BUFF[271] := -48, [3].Buffer.BUFF[272] := 83, [3].Buffer.BUFF[273] := 49, [3].Buffer.BUFF[274] := 57, [3].Buffer.BUFF[275] := 45, [3].Buffer.BUFF[276] := 66, [3].Buffer.BUFF[277] := 56, [3].Buffer.BUFF[278] := 45, [3].Buffer.BUFF[279] := 50, [3].Buffer.BUFF[280] := 48, [3].Buffer.BUFF[281] := 48, [3].Buffer.BUFF[282] := 49, [3].Buffer.BUFF[283] := 66, [3].Buffer.BUFF[285] := 45, [3].Buffer.BUFF[286] := 57, [3].Buffer.BUFF[287] := 57, [3].Buffer.BUFF[288] := 46, [3].Buffer.BUFF[289] := 48, [3].Buffer.BUFF[290] := 116, [3].Buffer.BUFF[291] := 32, [3].Buffer.BUFF[292] := 82, [3].Buffer.BUFF[294] := 3, [3].Buffer.BUFF[348] := 31, [3].Buffer.BUFF[352] := 2, [3].Buffer.BUFF[353] := 90, [3].Buffer.BUFF[354] := 48, [3].Buffer.BUFF[355] := -95, [3].Buffer.BUFF[356] := 1, [3].Buffer.BUFF[357] := 1, [3].Buffer.BUFF[358] := 78, [3].Buffer.BUFF[359] := -48, [3].Buffer.BUFF[360] := 83, [3].Buffer.BUFF[361] := 48, [3].Buffer.BUFF[362] := 45, [3].Buffer.BUFF[363] := 66, [3].Buffer.BUFF[364] := 49,
        [3].Buffer.BUFF[365] := 51, [3].Buffer.BUFF[366] := 57, [3].Buffer.BUFF[367] := 45, [3].Buffer.BUFF[368] := 51, [3].Buffer.BUFF[369] := 48, [3].Buffer.BUFF[370] := 49, [3].Buffer.BUFF[371] := 53, [3].Buffer.BUFF[374] := 45, [3].Buffer.BUFF[375] := 32, [3].Buffer.BUFF[376] := 51, [3].Buffer.BUFF[377] := 46, [3].Buffer.BUFF[378] := 48, [3].Buffer.BUFF[379] := 116, [3].Buffer.BUFF[380] := 82, [3].Buffer.BUFF[381] := 78, [3].Buffer.BUFF[382] := 3, [3].Buffer.BUFF[436] := 31, [3].Buffer.BUFF[440] := 2, [3].Buffer.BUFF[441] := 90, [3].Buffer.BUFF[442] := 48, [3].Buffer.BUFF[443] := -95, [3].Buffer.BUFF[444] := 1, [3].Buffer.BUFF[445] := 1, [3].Buffer.BUFF[446] := 78, [3].Buffer.BUFF[447] := -48, [3].Buffer.BUFF[448] := 66, [3].Buffer.BUFF[449] := 73, [3].Buffer.BUFF[450] := 78, [3].Buffer.BUFF[451] := 49, [3].Buffer.BUFF[452] := 32, [3].Buffer.BUFF[453] := 50, [3].Buffer.BUFF[454] := 48, [3].Buffer.BUFF[455] := 48, [3].Buffer.BUFF[456] := 49, [3].Buffer.BUFF[457] := 70, [3].Buffer.BUFF[459] := 45, [3].Buffer.BUFF[460] := 51, [3].Buffer.BUFF[461] := 48, [3].Buffer.BUFF[462] := 46, [3].Buffer.BUFF[463] := 48, [3].Buffer.BUFF[464] := 48, [3].Buffer.BUFF[465] := 116, [3].Buffer.BUFF[466] := 32, [3].Buffer.BUFF[467] := 32, [3].Buffer.BUFF[468] := 82, [3].Buffer.BUFF[469] := 98, [3].Buffer.BUFF[470] := 3, [3].Buffer.BUFF[471] := 82, [3].Buffer.BUFF[472] := 82, [3].Buffer.BUFF[473] := 82, [3].Buffer.BUFF[474] := 82, [3].Buffer.BUFF[475] := 82, [3].Buffer.BUFF[476] := 82, [3].Buffer.BUFF[477] := 82, [3].Buffer.BUFF[478] := 82, [3].Buffer.BUFF[479] := 82, [4].ToAddr.Family := 2, [4].ToAddr.Port := 8002, [4].ToAddr.Addr := 16#c101_017a, [4].Buffer.LEN := 31,
        [4].Buffer.BUFF[0] := 2, [4].Buffer.BUFF[1] := 90, [4].Buffer.BUFF[2] := 48, [4].Buffer.BUFF[3] := -95, [4].Buffer.BUFF[4] := 1, [4].Buffer.BUFF[5] := 1, [4].Buffer.BUFF[6] := 78, [4].Buffer.BUFF[7] := -48, [4].Buffer.BUFF[8] := 66, [4].Buffer.BUFF[9] := 73, [4].Buffer.BUFF[10] := 78, [4].Buffer.BUFF[11] := 58, [4].Buffer.BUFF[12] := 51, [4].Buffer.BUFF[13] := 52, [4].Buffer.BUFF[14] := 32, [4].Buffer.BUFF[15] := 50, [4].Buffer.BUFF[16] := 52, [4].Buffer.BUFF[17] := 49, [4].Buffer.BUFF[18] := 48, [4].Buffer.BUFF[21] := 45, [4].Buffer.BUFF[22] := 32, [4].Buffer.BUFF[23] := 54, [4].Buffer.BUFF[24] := 46, [4].Buffer.BUFF[25] := 48, [4].Buffer.BUFF[26] := 48, [4].Buffer.BUFF[27] := 116, [4].Buffer.BUFF[28] := 82, [4].Buffer.BUFF[29] := 57, [4].Buffer.BUFF[30] := 3, [4].Buffer.BUFF[84] := 31, [4].Buffer.BUFF[88] := 2, [4].Buffer.BUFF[89] := 90, [4].Buffer.BUFF[90] := 48, [4].Buffer.BUFF[91] := -95, [4].Buffer.BUFF[92] := 1, [4].Buffer.BUFF[93] := 1, [4].Buffer.BUFF[94] := 78, [4].Buffer.BUFF[95] := -48, [4].Buffer.BUFF[96] := 50, [4].Buffer.BUFF[97] := 48, [4].Buffer.BUFF[98] := 50, [4].Buffer.BUFF[99] := 54, [4].Buffer.BUFF[100] := 47, [4].Buffer.BUFF[101] := 48, [4].Buffer.BUFF[102] := 52, [4].Buffer.BUFF[103] := 47, [4].Buffer.BUFF[104] := 50, [4].Buffer.BUFF[105] := 57, [4].Buffer.BUFF[106] := 32, [4].Buffer.BUFF[107] := 32, [4].Buffer.BUFF[108] := 49, [4].Buffer.BUFF[109] := 48, [4].Buffer.BUFF[110] := 58, [4].Buffer.BUFF[111] := 50, [4].Buffer.BUFF[112] := 56, [4].Buffer.BUFF[113] := 58, [4].Buffer.BUFF[114] := 48, [4].Buffer.BUFF[115] := 55, [4].Buffer.BUFF[116] := 82, [4].Buffer.BUFF[117] := 2,
        [4].Buffer.BUFF[118] := 3, [4].Buffer.BUFF[172] := 31, [4].Buffer.BUFF[176] := 2, [4].Buffer.BUFF[177] := 90, [4].Buffer.BUFF[178] := 48, [4].Buffer.BUFF[179] := -95, [4].Buffer.BUFF[180] := 1, [4].Buffer.BUFF[181] := 1, [4].Buffer.BUFF[182] := 78, [4].Buffer.BUFF[183] := -48, [4].Buffer.BUFF[184] := 83, [4].Buffer.BUFF[185] := 49, [4].Buffer.BUFF[186] := 57, [4].Buffer.BUFF[187] := 45, [4].Buffer.BUFF[188] := 66, [4].Buffer.BUFF[189] := 56, [4].Buffer.BUFF[190] := 45, [4].Buffer.BUFF[191] := 50, [4].Buffer.BUFF[192] := 48, [4].Buffer.BUFF[193] := 48, [4].Buffer.BUFF[194] := 49, [4].Buffer.BUFF[195] := 66, [4].Buffer.BUFF[197] := 45, [4].Buffer.BUFF[198] := 57, [4].Buffer.BUFF[199] := 57, [4].Buffer.BUFF[200] := 46, [4].Buffer.BUFF[201] := 48, [4].Buffer.BUFF[202] := 116, [4].Buffer.BUFF[203] := 32, [4].Buffer.BUFF[204] := 82, [4].Buffer.BUFF[206] := 3, [4].Buffer.BUFF[260] := 31, [4].Buffer.BUFF[264] := 2, [4].Buffer.BUFF[265] := 90, [4].Buffer.BUFF[266] := 48, [4].Buffer.BUFF[267] := -95, [4].Buffer.BUFF[268] := 1, [4].Buffer.BUFF[269] := 1, [4].Buffer.BUFF[270] := 78, [4].Buffer.BUFF[271] := -48, [4].Buffer.BUFF[272] := 83, [4].Buffer.BUFF[273] := 48, [4].Buffer.BUFF[274] := 45, [4].Buffer.BUFF[275] := 66, [4].Buffer.BUFF[276] := 49, [4].Buffer.BUFF[277] := 51, [4].Buffer.BUFF[278] := 57, [4].Buffer.BUFF[279] := 45, [4].Buffer.BUFF[280] := 51, [4].Buffer.BUFF[281] := 48, [4].Buffer.BUFF[282] := 49, [4].Buffer.BUFF[283] := 53, [4].Buffer.BUFF[286] := 45, [4].Buffer.BUFF[287] := 32, [4].Buffer.BUFF[288] := 51, [4].Buffer.BUFF[289] := 46, [4].Buffer.BUFF[290] := 48, [4].Buffer.BUFF[291] := 116, [4].Buffer.BUFF[292] := 82, [4].Buffer.BUFF[293] := 78,
        [4].Buffer.BUFF[294] := 3, [4].Buffer.BUFF[348] := 8, [4].Buffer.BUFF[352] := 2, [4].Buffer.BUFF[353] := 90, [4].Buffer.BUFF[354] := 48, [4].Buffer.BUFF[355] := -88, [4].Buffer.BUFF[356] := 1, [4].Buffer.BUFF[357] := 1, [4].Buffer.BUFF[358] := -62, [4].Buffer.BUFF[359] := 3, [4].Buffer.BUFF[360] := 66, [4].Buffer.BUFF[361] := 73, [4].Buffer.BUFF[362] := 78, [4].Buffer.BUFF[363] := 49, [4].Buffer.BUFF[364] := 32, [4].Buffer.BUFF[365] := 50, [4].Buffer.BUFF[366] := 48, [4].Buffer.BUFF[367] := 48, [4].Buffer.BUFF[368] := 49, [4].Buffer.BUFF[369] := 70, [4].Buffer.BUFF[371] := 45, [4].Buffer.BUFF[372] := 51, [4].Buffer.BUFF[373] := 48, [4].Buffer.BUFF[374] := 46, [4].Buffer.BUFF[375] := 48, [4].Buffer.BUFF[376] := 48, [4].Buffer.BUFF[377] := 116, [4].Buffer.BUFF[378] := 32, [4].Buffer.BUFF[379] := 32, [4].Buffer.BUFF[380] := 82, [4].Buffer.BUFF[381] := 98, [4].Buffer.BUFF[382] := 3, [4].Buffer.BUFF[383] := 82, [4].Buffer.BUFF[384] := 82, [4].Buffer.BUFF[385] := 82, [4].Buffer.BUFF[386] := 82, [4].Buffer.BUFF[387] := 82, [4].Buffer.BUFF[388] := 82, [4].Buffer.BUFF[389] := 82, [4].Buffer.BUFF[390] := 82, [4].Buffer.BUFF[391] := 82, [4].Buffer.BUFF[392] := 82, [4].Buffer.BUFF[393] := 82, [4].Buffer.BUFF[394] := 82, [4].Buffer.BUFF[395] := 82, [4].Buffer.BUFF[396] := 82, [4].Buffer.BUFF[397] := 82, [4].Buffer.BUFF[398] := 82, [4].Buffer.BUFF[399] := 82, [4].Buffer.BUFF[400] := 82, [4].Buffer.BUFF[401] := 82, [4].Buffer.BUFF[402] := 82, [4].Buffer.BUFF[403] := 82, [4].Buffer.BUFF[404] := 82, [4].Buffer.BUFF[405] := 82, [4].Buffer.BUFF[406] := 82, [4].Buffer.BUFF[407] := 82, [4].Buffer.BUFF[408] := 82, [4].Buffer.BUFF[409] := 82, [4].Buffer.BUFF[410] := 82,
        [4].Buffer.BUFF[411] := 82, [4].Buffer.BUFF[412] := 82, [4].Buffer.BUFF[413] := 82, [4].Buffer.BUFF[414] := 82, [4].Buffer.BUFF[415] := -112, [4].Buffer.BUFF[416] := 3, [4].Buffer.BUFF[417] := 82, [4].Buffer.BUFF[418] := 82, [4].Buffer.BUFF[419] := 82, [4].Buffer.BUFF[420] := 82, [4].Buffer.BUFF[421] := 82, [4].Buffer.BUFF[422] := 82, [4].Buffer.BUFF[423] := 82, [4].Buffer.BUFF[424] := 82, [4].Buffer.BUFF[425] := 82, [4].Buffer.BUFF[426] := 82, [4].Buffer.BUFF[427] := 82, [4].Buffer.BUFF[428] := -62, [4].Buffer.BUFF[429] := 3, [4].Buffer.BUFF[430] := 3, [5].ToAddr.Family := 2, [5].ToAddr.Port := 8002, [5].ToAddr.Addr := 16#c101_017b, [5].Buffer.LEN := 31, [5].Buffer.BUFF[0] := 2, [5].Buffer.BUFF[1] := 90, [5].Buffer.BUFF[2] := 48, [5].Buffer.BUFF[3] := -95, [5].Buffer.BUFF[4] := 1, [5].Buffer.BUFF[5] := 1, [5].Buffer.BUFF[6] := 78, [5].Buffer.BUFF[7] := -48, [5].Buffer.BUFF[8] := 50, [5].Buffer.BUFF[9] := 48, [5].Buffer.BUFF[10] := 50, [5].Buffer.BUFF[11] := 54, [5].Buffer.BUFF[12] := 47, [5].Buffer.BUFF[13] := 48, [5].Buffer.BUFF[14] := 52, [5].Buffer.BUFF[15] := 47, [5].Buffer.BUFF[16] := 50, [5].Buffer.BUFF[17] := 57, [5].Buffer.BUFF[18] := 32, [5].Buffer.BUFF[19] := 32, [5].Buffer.BUFF[20] := 49, [5].Buffer.BUFF[21] := 48, [5].Buffer.BUFF[22] := 58, [5].Buffer.BUFF[23] := 50, [5].Buffer.BUFF[24] := 56, [5].Buffer.BUFF[25] := 58, [5].Buffer.BUFF[26] := 48, [5].Buffer.BUFF[27] := 56, [5].Buffer.BUFF[28] := 82, [5].Buffer.BUFF[29] := 13, [5].Buffer.BUFF[30] := 3, [5].Buffer.BUFF[84] := 31, [5].Buffer.BUFF[88] := 2, [5].Buffer.BUFF[89] := 90, [5].Buffer.BUFF[90] := 48, [5].Buffer.BUFF[91] := -95,
        [5].Buffer.BUFF[92] := 1, [5].Buffer.BUFF[93] := 1, [5].Buffer.BUFF[94] := 78, [5].Buffer.BUFF[95] := -48, [5].Buffer.BUFF[96] := 83, [5].Buffer.BUFF[97] := 49, [5].Buffer.BUFF[98] := 57, [5].Buffer.BUFF[99] := 45, [5].Buffer.BUFF[100] := 66, [5].Buffer.BUFF[101] := 56, [5].Buffer.BUFF[102] := 45, [5].Buffer.BUFF[103] := 50, [5].Buffer.BUFF[104] := 48, [5].Buffer.BUFF[105] := 48, [5].Buffer.BUFF[106] := 49, [5].Buffer.BUFF[107] := 66, [5].Buffer.BUFF[109] := 45, [5].Buffer.BUFF[110] := 57, [5].Buffer.BUFF[111] := 57, [5].Buffer.BUFF[112] := 46, [5].Buffer.BUFF[113] := 48, [5].Buffer.BUFF[114] := 116, [5].Buffer.BUFF[115] := 32, [5].Buffer.BUFF[116] := 82, [5].Buffer.BUFF[118] := 3, [5].Buffer.BUFF[172] := 31, [5].Buffer.BUFF[176] := 2, [5].Buffer.BUFF[177] := 90, [5].Buffer.BUFF[178] := 48, [5].Buffer.BUFF[179] := -95, [5].Buffer.BUFF[180] := 1, [5].Buffer.BUFF[181] := 1, [5].Buffer.BUFF[182] := 78, [5].Buffer.BUFF[183] := -48, [5].Buffer.BUFF[184] := 83, [5].Buffer.BUFF[185] := 48, [5].Buffer.BUFF[186] := 45, [5].Buffer.BUFF[187] := 66, [5].Buffer.BUFF[188] := 49, [5].Buffer.BUFF[189] := 51, [5].Buffer.BUFF[190] := 57, [5].Buffer.BUFF[191] := 45, [5].Buffer.BUFF[192] := 51, [5].Buffer.BUFF[193] := 48, [5].Buffer.BUFF[194] := 49, [5].Buffer.BUFF[195] := 53, [5].Buffer.BUFF[198] := 45, [5].Buffer.BUFF[199] := 32, [5].Buffer.BUFF[200] := 51, [5].Buffer.BUFF[201] := 46, [5].Buffer.BUFF[202] := 48, [5].Buffer.BUFF[203] := 116, [5].Buffer.BUFF[204] := 82, [5].Buffer.BUFF[205] := 78, [5].Buffer.BUFF[206] := 3, [5].Buffer.BUFF[260] := 31, [5].Buffer.BUFF[264] := 2, [5].Buffer.BUFF[265] := 90, [5].Buffer.BUFF[266] := 48, [5].Buffer.BUFF[267] := -95,
        [5].Buffer.BUFF[268] := 1, [5].Buffer.BUFF[269] := 1, [5].Buffer.BUFF[270] := 78, [5].Buffer.BUFF[271] := -48, [5].Buffer.BUFF[272] := 66, [5].Buffer.BUFF[273] := 73, [5].Buffer.BUFF[274] := 78, [5].Buffer.BUFF[275] := 49, [5].Buffer.BUFF[276] := 32, [5].Buffer.BUFF[277] := 50, [5].Buffer.BUFF[278] := 48, [5].Buffer.BUFF[279] := 48, [5].Buffer.BUFF[280] := 49, [5].Buffer.BUFF[281] := 70, [5].Buffer.BUFF[283] := 45, [5].Buffer.BUFF[284] := 51, [5].Buffer.BUFF[285] := 48, [5].Buffer.BUFF[286] := 46, [5].Buffer.BUFF[287] := 48, [5].Buffer.BUFF[288] := 48, [5].Buffer.BUFF[289] := 116, [5].Buffer.BUFF[290] := 32, [5].Buffer.BUFF[291] := 32, [5].Buffer.BUFF[292] := 82, [5].Buffer.BUFF[293] := 98, [5].Buffer.BUFF[294] := 3, [5].Buffer.BUFF[295] := 82, [5].Buffer.BUFF[296] := 82, [5].Buffer.BUFF[297] := 82, [5].Buffer.BUFF[298] := 82, [5].Buffer.BUFF[299] := 82, [5].Buffer.BUFF[300] := 82, [5].Buffer.BUFF[301] := 82, [5].Buffer.BUFF[302] := 82, [5].Buffer.BUFF[303] := 82, [5].Buffer.BUFF[304] := 82, [5].Buffer.BUFF[305] := 82, [5].Buffer.BUFF[306] := 82, [5].Buffer.BUFF[307] := 82, [5].Buffer.BUFF[308] := 82, [5].Buffer.BUFF[309] := 82, [5].Buffer.BUFF[310] := 82, [5].Buffer.BUFF[311] := 82, [5].Buffer.BUFF[312] := 82, [5].Buffer.BUFF[313] := 82, [5].Buffer.BUFF[314] := 82, [5].Buffer.BUFF[315] := 82, [5].Buffer.BUFF[316] := 82, [5].Buffer.BUFF[317] := 82, [5].Buffer.BUFF[318] := 82, [5].Buffer.BUFF[319] := 82, [5].Buffer.BUFF[320] := 82, [5].Buffer.BUFF[321] := 82, [5].Buffer.BUFF[322] := 82, [5].Buffer.BUFF[323] := 82, [5].Buffer.BUFF[324] := 82, [5].Buffer.BUFF[325] := 82, [5].Buffer.BUFF[326] := 82, [5].Buffer.BUFF[327] := -112, [5].Buffer.BUFF[328] := 3,
        [5].Buffer.BUFF[329] := 82, [5].Buffer.BUFF[330] := 82, [5].Buffer.BUFF[331] := 82, [5].Buffer.BUFF[332] := 82, [5].Buffer.BUFF[333] := 82, [5].Buffer.BUFF[334] := 82, [5].Buffer.BUFF[335] := 82, [5].Buffer.BUFF[336] := 82, [5].Buffer.BUFF[337] := 82, [5].Buffer.BUFF[338] := 82, [5].Buffer.BUFF[339] := 82, [5].Buffer.BUFF[340] := -62, [5].Buffer.BUFF[341] := 3, [5].Buffer.BUFF[342] := 3, [6].ToAddr.Family := 2, [6].ToAddr.Port := 8001, [6].ToAddr.Addr := 16#c101_017c, [6].Buffer.LEN := 31, [6].Buffer.BUFF[0] := 2, [6].Buffer.BUFF[1] := 90, [6].Buffer.BUFF[2] := 48, [6].Buffer.BUFF[3] := -95, [6].Buffer.BUFF[4] := 1, [6].Buffer.BUFF[5] := 1, [6].Buffer.BUFF[6] := 78, [6].Buffer.BUFF[7] := -48, [6].Buffer.BUFF[8] := 83, [6].Buffer.BUFF[9] := 49, [6].Buffer.BUFF[10] := 57, [6].Buffer.BUFF[11] := 45, [6].Buffer.BUFF[12] := 66, [6].Buffer.BUFF[13] := 56, [6].Buffer.BUFF[14] := 45, [6].Buffer.BUFF[15] := 50, [6].Buffer.BUFF[16] := 48, [6].Buffer.BUFF[17] := 48, [6].Buffer.BUFF[18] := 49, [6].Buffer.BUFF[19] := 66, [6].Buffer.BUFF[21] := 45, [6].Buffer.BUFF[22] := 57, [6].Buffer.BUFF[23] := 57, [6].Buffer.BUFF[24] := 46, [6].Buffer.BUFF[25] := 48, [6].Buffer.BUFF[26] := 116, [6].Buffer.BUFF[27] := 32, [6].Buffer.BUFF[28] := 82, [6].Buffer.BUFF[30] := 3, [6].Buffer.BUFF[84] := 31, [6].Buffer.BUFF[88] := 2, [6].Buffer.BUFF[89] := 90, [6].Buffer.BUFF[90] := 48, [6].Buffer.BUFF[91] := -95, [6].Buffer.BUFF[92] := 1, [6].Buffer.BUFF[93] := 1, [6].Buffer.BUFF[94] := 78, [6].Buffer.BUFF[95] := -48, [6].Buffer.BUFF[96] := 83, [6].Buffer.BUFF[97] := 48, [6].Buffer.BUFF[98] := 45, [6].Buffer.BUFF[99] := 66,
        [6].Buffer.BUFF[100] := 49, [6].Buffer.BUFF[101] := 51, [6].Buffer.BUFF[102] := 57, [6].Buffer.BUFF[103] := 45, [6].Buffer.BUFF[104] := 51, [6].Buffer.BUFF[105] := 48, [6].Buffer.BUFF[106] := 49, [6].Buffer.BUFF[107] := 53, [6].Buffer.BUFF[110] := 45, [6].Buffer.BUFF[111] := 32, [6].Buffer.BUFF[112] := 51, [6].Buffer.BUFF[113] := 46, [6].Buffer.BUFF[114] := 48, [6].Buffer.BUFF[115] := 116, [6].Buffer.BUFF[116] := 82, [6].Buffer.BUFF[117] := 78, [6].Buffer.BUFF[118] := 3, [6].Buffer.BUFF[172] := 31, [6].Buffer.BUFF[176] := 2, [6].Buffer.BUFF[177] := 90, [6].Buffer.BUFF[178] := 48, [6].Buffer.BUFF[179] := -95, [6].Buffer.BUFF[180] := 1, [6].Buffer.BUFF[181] := 1, [6].Buffer.BUFF[182] := 78, [6].Buffer.BUFF[183] := -48, [6].Buffer.BUFF[184] := 66, [6].Buffer.BUFF[185] := 73, [6].Buffer.BUFF[186] := 78, [6].Buffer.BUFF[187] := 49, [6].Buffer.BUFF[188] := 32, [6].Buffer.BUFF[189] := 50, [6].Buffer.BUFF[190] := 48, [6].Buffer.BUFF[191] := 48, [6].Buffer.BUFF[192] := 49, [6].Buffer.BUFF[193] := 70, [6].Buffer.BUFF[195] := 45, [6].Buffer.BUFF[196] := 51, [6].Buffer.BUFF[197] := 48, [6].Buffer.BUFF[198] := 46, [6].Buffer.BUFF[199] := 48, [6].Buffer.BUFF[200] := 48, [6].Buffer.BUFF[201] := 116, [6].Buffer.BUFF[202] := 32, [6].Buffer.BUFF[203] := 32, [6].Buffer.BUFF[204] := 82, [6].Buffer.BUFF[205] := 98, [6].Buffer.BUFF[206] := 3, [6].Buffer.BUFF[207] := 82, [6].Buffer.BUFF[208] := 82, [6].Buffer.BUFF[209] := 82, [6].Buffer.BUFF[210] := 82, [6].Buffer.BUFF[211] := 82, [6].Buffer.BUFF[212] := 82, [6].Buffer.BUFF[213] := 82, [6].Buffer.BUFF[214] := 82, [6].Buffer.BUFF[215] := 82, [6].Buffer.BUFF[216] := 82, [6].Buffer.BUFF[217] := 82, [6].Buffer.BUFF[218] := 82,
        [6].Buffer.BUFF[219] := 82, [6].Buffer.BUFF[220] := 82, [6].Buffer.BUFF[221] := 82, [6].Buffer.BUFF[222] := 82, [6].Buffer.BUFF[223] := 82, [6].Buffer.BUFF[224] := 82, [6].Buffer.BUFF[225] := 82, [6].Buffer.BUFF[226] := 82, [6].Buffer.BUFF[227] := 82, [6].Buffer.BUFF[228] := 82, [6].Buffer.BUFF[229] := 82, [6].Buffer.BUFF[230] := 82, [6].Buffer.BUFF[231] := 82, [6].Buffer.BUFF[232] := 82, [6].Buffer.BUFF[233] := 82, [6].Buffer.BUFF[234] := 82, [6].Buffer.BUFF[235] := 82, [6].Buffer.BUFF[236] := 82, [6].Buffer.BUFF[237] := 82, [6].Buffer.BUFF[238] := 82, [6].Buffer.BUFF[239] := -112, [6].Buffer.BUFF[240] := 3, [6].Buffer.BUFF[241] := 82, [6].Buffer.BUFF[242] := 82, [6].Buffer.BUFF[243] := 82, [6].Buffer.BUFF[244] := 82, [6].Buffer.BUFF[245] := 82, [6].Buffer.BUFF[246] := 82, [6].Buffer.BUFF[247] := 82, [6].Buffer.BUFF[248] := 82, [6].Buffer.BUFF[249] := 82, [6].Buffer.BUFF[250] := 82, [6].Buffer.BUFF[251] := 82, [6].Buffer.BUFF[252] := -62, [6].Buffer.BUFF[253] := 3, [6].Buffer.BUFF[254] := 3, [7].ToAddr.Family := 2, [7].ToAddr.Port := 8001, [7].ToAddr.Addr := 16#c101_017d, [7].Buffer.LEN := 31, [7].Buffer.BUFF[0] := 2, [7].Buffer.BUFF[1] := 90, [7].Buffer.BUFF[2] := 48, [7].Buffer.BUFF[3] := -95, [7].Buffer.BUFF[4] := 1, [7].Buffer.BUFF[5] := 1, [7].Buffer.BUFF[6] := 78, [7].Buffer.BUFF[7] := -48, [7].Buffer.BUFF[8] := 83, [7].Buffer.BUFF[9] := 48, [7].Buffer.BUFF[10] := 45, [7].Buffer.BUFF[11] := 66, [7].Buffer.BUFF[12] := 49, [7].Buffer.BUFF[13] := 51, [7].Buffer.BUFF[14] := 57, [7].Buffer.BUFF[15] := 45, [7].Buffer.BUFF[16] := 51, [7].Buffer.BUFF[17] := 48, [7].Buffer.BUFF[18] := 49, [7].Buffer.BUFF[19] := 53,
        [7].Buffer.BUFF[22] := 45, [7].Buffer.BUFF[23] := 32, [7].Buffer.BUFF[24] := 51, [7].Buffer.BUFF[25] := 46, [7].Buffer.BUFF[26] := 48, [7].Buffer.BUFF[27] := 116, [7].Buffer.BUFF[28] := 82, [7].Buffer.BUFF[29] := 78, [7].Buffer.BUFF[30] := 3, [7].Buffer.BUFF[84] := 31, [7].Buffer.BUFF[88] := 2, [7].Buffer.BUFF[89] := 90, [7].Buffer.BUFF[90] := 48, [7].Buffer.BUFF[91] := -95, [7].Buffer.BUFF[92] := 1, [7].Buffer.BUFF[93] := 1, [7].Buffer.BUFF[94] := 78, [7].Buffer.BUFF[95] := -48, [7].Buffer.BUFF[96] := 66, [7].Buffer.BUFF[97] := 73, [7].Buffer.BUFF[98] := 78, [7].Buffer.BUFF[99] := 49, [7].Buffer.BUFF[100] := 32, [7].Buffer.BUFF[101] := 50, [7].Buffer.BUFF[102] := 48, [7].Buffer.BUFF[103] := 48, [7].Buffer.BUFF[104] := 49, [7].Buffer.BUFF[105] := 70, [7].Buffer.BUFF[107] := 45, [7].Buffer.BUFF[108] := 51, [7].Buffer.BUFF[109] := 48, [7].Buffer.BUFF[110] := 46, [7].Buffer.BUFF[111] := 48, [7].Buffer.BUFF[112] := 48, [7].Buffer.BUFF[113] := 116, [7].Buffer.BUFF[114] := 32, [7].Buffer.BUFF[115] := 32, [7].Buffer.BUFF[116] := 82, [7].Buffer.BUFF[117] := 98, [7].Buffer.BUFF[118] := 3, [7].Buffer.BUFF[119] := 82, [7].Buffer.BUFF[120] := 82, [7].Buffer.BUFF[121] := 82, [7].Buffer.BUFF[122] := 82, [7].Buffer.BUFF[123] := 82, [7].Buffer.BUFF[124] := 82, [7].Buffer.BUFF[125] := 82, [7].Buffer.BUFF[126] := 82, [7].Buffer.BUFF[127] := 82, [7].Buffer.BUFF[128] := 82, [7].Buffer.BUFF[129] := 82, [7].Buffer.BUFF[130] := 82, [7].Buffer.BUFF[131] := 82, [7].Buffer.BUFF[132] := 82, [7].Buffer.BUFF[133] := 82, [7].Buffer.BUFF[134] := 82, [7].Buffer.BUFF[135] := 82, [7].Buffer.BUFF[136] := 82, [7].Buffer.BUFF[137] := 82, [7].Buffer.BUFF[138] := 82,
        [7].Buffer.BUFF[139] := 82, [7].Buffer.BUFF[140] := 82, [7].Buffer.BUFF[141] := 82, [7].Buffer.BUFF[142] := 82, [7].Buffer.BUFF[143] := 82, [7].Buffer.BUFF[144] := 82, [7].Buffer.BUFF[145] := 82, [7].Buffer.BUFF[146] := 82, [7].Buffer.BUFF[147] := 82, [7].Buffer.BUFF[148] := 82, [7].Buffer.BUFF[149] := 82, [7].Buffer.BUFF[150] := 82, [7].Buffer.BUFF[151] := -112, [7].Buffer.BUFF[152] := 3, [7].Buffer.BUFF[153] := 82, [7].Buffer.BUFF[154] := 82, [7].Buffer.BUFF[155] := 82, [7].Buffer.BUFF[156] := 82, [7].Buffer.BUFF[157] := 82, [7].Buffer.BUFF[158] := 82, [7].Buffer.BUFF[159] := 82, [7].Buffer.BUFF[160] := 82, [7].Buffer.BUFF[161] := 82, [7].Buffer.BUFF[162] := 82, [7].Buffer.BUFF[163] := 82, [7].Buffer.BUFF[164] := -62, [7].Buffer.BUFF[165] := 3, [7].Buffer.BUFF[166] := 3, [8].ToAddr.Family := 2, [8].ToAddr.Port := 8002, [8].ToAddr.Addr := 16#c101_017e, [8].Buffer.LEN := 31, [8].Buffer.BUFF[0] := 2, [8].Buffer.BUFF[1] := 90, [8].Buffer.BUFF[2] := 48, [8].Buffer.BUFF[3] := -95, [8].Buffer.BUFF[4] := 1, [8].Buffer.BUFF[5] := 1, [8].Buffer.BUFF[6] := 78, [8].Buffer.BUFF[7] := -48, [8].Buffer.BUFF[8] := 66, [8].Buffer.BUFF[9] := 73, [8].Buffer.BUFF[10] := 78, [8].Buffer.BUFF[11] := 49, [8].Buffer.BUFF[12] := 32, [8].Buffer.BUFF[13] := 50, [8].Buffer.BUFF[14] := 48, [8].Buffer.BUFF[15] := 48, [8].Buffer.BUFF[16] := 49, [8].Buffer.BUFF[17] := 70, [8].Buffer.BUFF[19] := 45, [8].Buffer.BUFF[20] := 51, [8].Buffer.BUFF[21] := 48, [8].Buffer.BUFF[22] := 46, [8].Buffer.BUFF[23] := 48, [8].Buffer.BUFF[24] := 48, [8].Buffer.BUFF[25] := 116, [8].Buffer.BUFF[26] := 32, [8].Buffer.BUFF[27] := 32, [8].Buffer.BUFF[28] := 82,
        [8].Buffer.BUFF[29] := 98, [8].Buffer.BUFF[30] := 3, [8].Buffer.BUFF[31] := 82, [8].Buffer.BUFF[32] := 82, [8].Buffer.BUFF[33] := 82, [8].Buffer.BUFF[34] := 82, [8].Buffer.BUFF[35] := 82, [8].Buffer.BUFF[36] := 82, [8].Buffer.BUFF[37] := 82, [8].Buffer.BUFF[38] := 82, [8].Buffer.BUFF[39] := 82, [8].Buffer.BUFF[40] := 82, [8].Buffer.BUFF[41] := 82, [8].Buffer.BUFF[42] := 82, [8].Buffer.BUFF[43] := 82, [8].Buffer.BUFF[44] := 82, [8].Buffer.BUFF[45] := 82, [8].Buffer.BUFF[46] := 82, [8].Buffer.BUFF[47] := 82, [8].Buffer.BUFF[48] := 82, [8].Buffer.BUFF[49] := 82, [8].Buffer.BUFF[50] := 82, [8].Buffer.BUFF[51] := 82, [8].Buffer.BUFF[52] := 82, [8].Buffer.BUFF[53] := 82, [8].Buffer.BUFF[54] := 82, [8].Buffer.BUFF[55] := 82, [8].Buffer.BUFF[56] := 82, [8].Buffer.BUFF[57] := 82, [8].Buffer.BUFF[58] := 82, [8].Buffer.BUFF[59] := 82, [8].Buffer.BUFF[60] := 82, [8].Buffer.BUFF[61] := 82, [8].Buffer.BUFF[62] := 82, [8].Buffer.BUFF[63] := -112, [8].Buffer.BUFF[64] := 3, [8].Buffer.BUFF[65] := 82, [8].Buffer.BUFF[66] := 82, [8].Buffer.BUFF[67] := 82, [8].Buffer.BUFF[68] := 82, [8].Buffer.BUFF[69] := 82, [8].Buffer.BUFF[70] := 82, [8].Buffer.BUFF[71] := 82, [8].Buffer.BUFF[72] := 82, [8].Buffer.BUFF[73] := 82, [8].Buffer.BUFF[74] := 82, [8].Buffer.BUFF[75] := 82, [8].Buffer.BUFF[76] := -62, [8].Buffer.BUFF[77] := 3, [8].Buffer.BUFF[78] := 3);
   Now : DateTime_Type := (Year := 2026, Month := 6, Day := 5, Hour := 8, Minute := 19, Second := 56, Microseconds := 381885);
   rcp_Auto : ALIAS FOR SYS_E.AUTO;
   rcp_Batch : DINT;
   rcp_Batch_OK : BOOL;
   rcp_Batch_Start : BOOL;
   rcp_Big : Part_Type := (Bin[0] := 1, Bin[1] := 2, Bin_Index[1] := 1, Number[0] := 730000570, Number[1] := 730000930, SetWeight[0] := 300.0, SetWeight[1] := 600.0);
        .Bin   // 大磅原料Bin號
        .Bin_Index   // 大磅原料桶指標
        .Number   // 大磅原料代號
        .SetWeight   // 大磅設重
        .RealWeight   // 大磅實重
        .ErrorWeight   // 大磅誤差重量
   rcp_Big_Add : BOOL;
   rcp_Big_Add_Cmd : BOOL;
   rcp_Big_Add_Skip : BOOL;
   rcp_Big_Bin : Bin_Raw[20] := ([0].LL := 1, [0].Bin := 1, [0].Bin_ID := 1, [0].Fall := 34.0, [0].Hi_Speed := 50, [0].Low_Speed := 10, [0].Low_Weight := 25, [0].Number := 730000570, [0].N0 := '1011', [1].LL := 1, [1].Bin := 2, [1].Bin_ID := 2, [1].Fall := 26.0, [1].Hi_Speed := 60, [1].Low_Speed := 20, [1].Low_Weight := 50, [1].Number := 730000930, [1].N0 := '2001', [1].N1 := 'F$00@$D0', [2].LL := 1, [2].YL := 1, [2].LS := 1, [2].Bin := 3, [2].Bin_ID := 3, [2].Fall := 10.0, [2].Hi_Speed := 60, [2].Low_Speed := 20, [2].Low_Weight := 50, [2].Number := 730002880, [2].N0 := '2024', [3].Bin := 4, [3].Bin_ID := 4, [3].Fall := 43.0, [3].Hi_Speed := 60, [3].Low_Speed := 20, [3].Low_Weight := 50, [3].Number := 770000871, [3].N0 := '1002', [3].N1 := 'Q$00$E6_', [4].LL := 1, [4].Bin := 5, [4].Bin_ID := 5, [4].Fall := 4.0, [4].Hi_Speed := 60, [4].Low_Speed := 20, [4].Low_Weight := 50, [4].Number := 730000550, [4].N0 := '1003', [4].N1 := 'B$00A$86', [5].LL := 1, [5].Bin := 6, [5].Bin_ID := 6, [5].Fall := 4.0, [5].Hi_Speed := 60, [5].Low_Speed := 20, [5].Low_Weight := 50, [5].Number := 730001060, [5].N0 := '2308', [5].N1 := 'A$00F$00', [6].Bin := 7,
        [6].Bin_ID := 7, [6].Fall := 10.0, [6].Hi_Speed := 60, [6].Low_Speed := 20, [6].Low_Weight := 50, [6].Number := 770002890, [6].N0 := '1001', [6].N1 := 'B$00[$01', [7].Bin := 8, [7].Bin_ID := 8, [7].Fall := 12.0, [7].Hi_Speed := 20, [7].Low_Speed := 10, [7].Low_Weight := 10, [7].Number := 730004080, [7].N0 := '2700', [8].Bin := 9, [8].Bin_ID := 9, [8].Fall := 4.0, [8].Hi_Speed := 60, [8].Low_Speed := 20, [8].Low_Weight := 50, [8].Number := 730003020, [8].N0 := '3001', [8].N1 := 'M$00$$$CE', [9].Bin := 10, [9].Bin_ID := 10, [9].Fall := 20.0, [9].Hi_Speed := 60, [9].Low_Speed := 20, [9].Low_Weight := 50, [9].Number := 730000970, [9].N0 := '2018', [9].N1 := 'A$00$7F$16', [10].Disable := 1, [10].Bin := 11, [10].Bin_ID := 11, [10].Fall := 5.0, [10].Hi_Speed := 60, [10].Low_Speed := 20, [10].Low_Weight := 50, [10].Number := 730000780, [10].N0 := '2001', [10].N1 := 'B$00$C0$B3', [11].Bin := 12, [11].Bin_ID := 12, [11].Fall := 8.0, [11].Hi_Speed := 60, [11].Low_Speed := 20, [11].Low_Weight := 50, [11].Number := 730001930, [11].N0 := '3123', [12].Bin := 13, [12].Bin_ID := 13, [12].Fall := 42.0, [12].Hi_Speed := 50, [12].Low_Speed := 10, [12].Low_Weight := 50, [12].Number := 730000900, [12].N0 := '1002',
        [12].N1 := 'V$00$12F', [13].Bin := 14, [13].Bin_ID := 14, [13].Fall := 13.0, [13].Hi_Speed := 45, [13].Low_Speed := 10, [13].Low_Weight := 60, [13].Number := 730000871, [13].N0 := '1002', [13].N1 := 'Q$00$0FF', [14].Bin := 15, [14].Bin_ID := 15, [14].Fall := 3.0, [14].Hi_Speed := 60, [14].Low_Speed := 20, [14].Low_Weight := 50, [14].Number := 730004120, [14].N0 := '1003', [14].N1 := 'E$008$C6', [15].Bin := 16, [15].Bin_ID := 16, [15].Fall := 4.0, [15].Hi_Speed := 60, [15].Low_Speed := 20, [15].Low_Weight := 50, [15].Number := 770002910, [15].N0 := '2002', [15].N1 := 'B$00$CEd', [16].Bin := 29, [16].Bin_ID := 104, [16].Fall := 6.0, [16].Hi_Speed := 50, [16].Low_Speed := 20, [16].Low_Weight := 50, [16].Number := 730002870, [16].N0 := '2029', [17].LL := 1, [17].Disable := 1, [17].Bin := 56, [17].Bin_ID := 56, [17].Fall := 3.0, [17].Hi_Speed := 35, [17].Low_Speed := 20, [17].Low_Weight := 30, [17].Number := 730003940, [17].N0 := '2310', [18].Hi_Speed := 80, [18].Low_Speed := 20, [18].Low_Weight := 5, [19].Hi_Speed := 80, [19].Low_Speed := 20, [19].Low_Weight := 5);
   rcp_Big_Bridge : BOOL;
   rcp_Big_Bridge_skip : BOOL;
   rcp_Big_Continue : BOOL;
   rcp_Big_Pause : BOOL := 1;
   rcp_Big_Run : BOOL;
   rcp_Big_Scale : REAL;
   rcp_Big_Speed : DINT;
   rcp_BigBin_Change : DINT := 10000;
   rcp_BigLastID : DINT := 2;
   rcp_BigLastID1 : DINT;
   rcp_Cancel_Pause : BOOL;
   rcp_class : DINT;
   rcp_Clear : BOOL;
   rcp_Dest_Bin : DINT;
   rcp_Hand : Part_Type_Hand := (Number[0] := 123456789, SetWeight[0] := 15.0, ErrorWeight[10] := -1.5e-43, ErrorWeight[11] := -1.e-44, ErrorWeight[12] := 1.4174465e-38, ErrorWeight[13] := 2.8669248e-37, ErrorWeight[14] := 4.316543e-39, ErrorWeight[15] := 6.e-45, ErrorWeight[17] := -1.e-44, ErrorWeight[18] := -1.e-44, ErrorWeight[19] := 1.4174465e-38, ErrorWeight[20] := 2.8670208e-37, ErrorWeight[21] := 4.224716e-39, ErrorWeight[22] := 6.e-45, ErrorWeight[23] := 1.0, ErrorWeight[24] := -1.e-44, ErrorWeight[25] := -1.3e-44, ErrorWeight[26] := 1.4174465e-38, ErrorWeight[27] := 2.867027e-37, ErrorWeight[28] := 4.18408e-39, ErrorWeight[29] := 1.7e-44);
   rcp_Hand_Index : DINT := 1;
   rcp_Hand_PB : BOOL;
   rcp_Hand_Run : BOOL;
   rcp_Hand_Scale : REAL;
   rcp_Hand_Total : DINT := 60;
   rcp_Mult : REAL := 3.0;
   rcp_Recipe : Recipe_Type := (Number[0] := 'Test', BatchSet := 2, Date := 20260605, pNumber[0] := 730000570, pNumber[1] := 730000930, pNumber[2] := 123456789, pSetWeight[0] := 300.0, pSetWeight[1] := 600.0, pSetWeight[2] := 15.0);
   rcp_Recipe_pNumber : DINT[20] := ([0] := 730000570, [1] := 730000930, [2] := 123456789);
   rcp_Recipe_Power_Reset : BOOL := 1;
   rcp_Recipe_pSetweight : REAL[20] := ([0] := 100.0, [1] := 200.0, [2] := 5.0);
   rcp_Recipe_Reset : BOOL;
   rcp_Report_Bin : INT[66] := ([0] := 25, [1] := 26, [2] := 17, [3] := 11, [4] := 14, [5] := 18, [6] := 101, [7] := 38, [8] := 19, [9] := 41, [10] := 40, [11] := 99, [12] := 99, [13] := 99, [14] := 99, [15] := 351, [16] := 352, [17] := 353, [18] := 356, [40] := 3, [41] := 55, [42] := 13, [44] := 1, [45] := 61, [46] := 29556, [47] := 21605, [52] := 9981, [53] := 309);
        [0]   // 大磅配方Bin
        [20]   // 大磅手動Bin
        [25]   // 小磅配方Bin
        [40]   // 配方開始HH
        [41]   // 配方開始MM
        [42]   // 配方開始SS
        [43]   // 班別(1=A,2=B,3=C)
        [44]   // Batch
        [45]   // Dest Bin
        [46]   // 配方代號
        [50]   // 配方日期
        [52]   // 配方說明
   rcp_Report_Log : BOOL;
   rcp_Report_Number : DINT[60] := ([0] := '+$82$EE$04', [1] := '+$82$ED$E7', [2] := '+$82$FAp', [3] := '+$82$EE"', [4] := '+$82$EC$A6', [5] := '+$82$F6L', [6] := '+$82$F8,', [7] := '+$82$F1$F6', [8] := '+$82$F7$F0', [9] := '+$83$00V', [10] := '+$82$EA$8A', [11] := '+$82$F1$E2', [12] := '+$82$F2$D2', [13] := '+$82$EBR', [14] := '+$82$F2$BE', [15] := '+$82$EB>', [16] := '+$82$F3$E0', [17] := '+$82$F0$A2', [18] := '+$82$EBp', [40] := '+$82$F7F', [41] := '+$82$F1$CE', [42] := '+$83$01$AA');
        [0]   // 大磅配方原料代號
   rcp_Report_RealWeight : REAL[60] := ([0] := 600.0, [1] := 682.0, [2] := 31.0, [3] := 592.0, [4] := 210.0, [5] := 57.0, [6] := 240.0, [7] := 360.0, [8] := 59.0, [9] := 29.0, [10] := 24.0, [11] := 44.2, [12] := 2.5, [13] := 0.6, [14] := 44.8, [15] := 11.417572, [16] := 5.98822, [17] := 6.0737915, [18] := 5.359665, [40] := 23.6, [41] := 11.299999, [42] := 0.3999977);
   rcp_Report_SetWeight : REAL[60] := ([0] := 600.0, [1] := 683.4, [2] := 30.0, [3] := 588.0, [4] := 210.0, [5] := 58.5, [6] := 240.0, [7] := 360.0, [8] := 60.0, [9] := 30.0, [10] := 25.800001, [11] := 45.0, [12] := 2.4, [13] := 0.6, [14] := 45.0, [15] := 11.4, [16] := 6.0, [17] := 6.0, [18] := 5.3999996, [40] := 24.0, [41] := 12.900001, [42] := 0.6);
   rcp_RUN : BOOL;
   rcp_Scale_Lock : BOOL := 1;
   rcp_Scale_Open : BOOL;
   rcp_schedule : Recipe_Type[11] := ([0].Number[0] := 'Test', [0].BatchSet := 2, [0].Date := 20260605, [0].pNumber[0] := 730000570, [0].pNumber[1] := 730000930, [0].pNumber[2] := 123456789, [0].pSetWeight[0] := 100.0, [0].pSetWeight[1] := 200.0, [0].pSetWeight[2] := 5.0);
   rcp_schedule_Index : DINT;
   rcp_Schedule_INPUT : BOOL;
   rcp_ScheduleLog : ScheduleLog[10] := ([1].Number[0] := 'Test', [1].StartTime := 605124577, [1].Batch := 2, [2].Number[0] := 'Test', [2].StartTime := 605131534, [2].Batch := 2, [3].Number[0] := 'Test', [3].StartTime := 605134553, [3].Batch := 2, [4].Number[0] := 'Test', [4].StartTime := 605141111, [4].Batch := 2, [5].Number[0] := 'Test', [5].StartTime := 605293589, [5].Batch := 2, [6].Number[0] := 'Test', [6].StartTime := 605294692, [6].Batch := 2, [7].Number[0] := 'Test', [7].StartTime := 605295253, [7].Batch := 3, [8].Number[0] := 'Test', [8].StartTime := 605297595, [8].Batch := 3, [9].Number[0] := 'Test', [9].StartTime := 605298284, [9].Batch := 2);
   rcp_Set_Pause : BOOL;
   SCALE_SIMULATE : BOOL := 1;
   STS : INT[100] := ([0] := 17, [23] := 5, [33] := 11, [34] := 4, [35] := 11, [36] := 11, [37] := 11, [38] := 11, [39] := 11, [40] := 11, [41] := 11, [42] := 11, [43] := 11, [44] := 11, [45] := 11, [46] := 11, [47] := 11, [48] := 11, [49] := 11, [50] := 11, [52] := 5, [53] := 5, [54] := 5, [55] := 11, [56] := 4);
   SYS : System_Common := (Simulate := 1, FlashFast := 1, PSH := 1, PSL := 1, DAY := 5, Day_Hour := 5, Year := 10000, MMDDHHMMs := 605299963);
   SYS_B : Sys_Data := (SIMULATE := 1, FlashFast := 1, Day := 5, Day_Hour := 5, Year := 10000, MSG_ID := 1, MMDDHHMMS := 605299963, ActLog[16].Time := 605304919, ActLog[16].STS := 10503, ActLog[17].Time := 605304919, ActLog[17].STS := 10303, ActLog[18].Time := 605219446, ActLog[18].STS := 10029, ActLog[19].Time := 605219557, ActLog[19].STS := 10017);
   SYS_B_DELAY : TIMER := (PRE := 10000);
   SYS_D : Sys_Data := (SIMULATE := 1, FlashFast := 1, Day := 5, Day_Hour := 5, Year := 10000, MSG_ID := 1, MMDDHHMMS := 605299963);
   SYS_E : Sys_Data := (MC := 1, AUTO := 1, SIMULATE := 1, FlashFast := 1, Power := 1, Flag := 1, Day := 5, Day_Hour := 5, Year := 10000, MSG_ID := 4, MMDDHHMMS := 605299963, ActLog[12].Time := 605361396, ActLog[12].STS := 10029, ActLog[13].Time := 605361663, ActLog[13].STS := 10018, ActLog[14].Time := 605124658, ActLog[14].STS := 10029, ActLog[15].Time := 605124716, ActLog[15].STS := 10017, ActLog[16].Time := 605131243, ActLog[16].STS := 10029, ActLog[17].Time := 605131269, ActLog[17].STS := 10017, ActLog[18].Time := 605293313, ActLog[18].STS := 10029, ActLog[19].Time := 605293392, ActLog[19].STS := 10017);
   SYS_F : Sys_Data := (SIMULATE := 1, FlashFast := 1, Day := 5, Day_Hour := 5, Year := 10000, MSG_ID := 1, MMDDHHMMS := 605299963);
END_VAR

PROGRAM LED_UDP   (* main routine MainRoutine *)
VAR
   DateTime : DateTime_String;
   HS1 : STRING := '100.0';
   Led_CMD : LED_CMD;
   Led_Min_Interval : TIMER[16] := ([0].PRE := 500, [0].ACC := 500, [1].PRE := 2000, [1].ACC := 201, [1].TT := 1, [1].DN := 1, [2].PRE := 500, [2].ACC := 98, [2].TT := 1, [2].DN := 1, [3].PRE := 500, [3].ACC := 150, [3].TT := 1, [3].DN := 1, [4].PRE := 500, [4].ACC := 149, [4].TT := 1, [4].DN := 1, [5].PRE := 800, [5].ACC := 556, [5].TT := 1, [5].DN := 1, [6].PRE := 800, [6].ACC := 98, [6].TT := 1, [6].DN := 1, [7].PRE := 500, [7].ACC := 148, [7].TT := 1, [7].DN := 1, [8].PRE := 500, [8].ACC := 201, [8].TT := 1, [8].DN := 1);
   Led_Prev_strout : STRING[16] := ([0] := '$02Z0$A1$01$01N$D0770031390d 5-3      RP$03', [1] := '$02Z0$A1$01$01N$D02026/04/29  10:28:16R$02$03', [2] := '$02Z0$A1$01$01N$D0730000600  100.0 Kg R6$03', [3] := '$02Z0$A1$01$01N$D0BIN:41 3016E 5.00 t RS$03', [4] := '$02Z0$A1$01$01N$D0BIN:34 2410$00$00- 6.00tR9$03', [5] := '$02Z0$A1$01$01N$D02026/04/29  10:28:15R$01$03', [6] := '$02Z0$A1$01$01N$D0S19-B8-2001B$00-99.0t R$00$03', [7] := '$02Z0$A1$01$01N$D0S0-B139-3015$00$00- 3.0tRN$03', [8] := '$02Z0$A1$01$01N$D0BIN1 2001F$00-30.00t  Rb$03');
   Led_ReSend_T : TIMER[16] := ([0].PRE := 1000, [1].PRE := 1000, [1].ACC := 103, [1].EN := 1, [1].TT := 1, [2].PRE := 1000, [2].EN := 1, [2].TT := 1, [3].PRE := 1000, [3].ACC := 51, [3].EN := 1, [3].TT := 1, [4].PRE := 1000, [4].ACC := 51, [4].EN := 1, [4].TT := 1, [5].PRE := 1000, [5].ACC := 458, [5].EN := 1, [5].TT := 1, [6].PRE := 1000, [6].EN := 1, [6].TT := 1, [7].PRE := 1000, [7].ACC := 50, [7].EN := 1, [7].TT := 1, [8].PRE := 1000, [8].ACC := 103, [8].EN := 1, [8].TT := 1);
   Led_SendHead : STRING := 'Z0$A1$01$01N$D0';
   Led_SendLast : STRING := 'R';
   Led_SendLine : STRING := 'Z0$A8$01$01';
   Led_SendLine_T : TIMER[16] := ([0].PRE := 60000, [0].ACC := 25312, [0].EN := 1, [0].TT := 1, [1].PRE := 3000, [1].ACC := 2542, [1].EN := 1, [1].TT := 1, [2].PRE := 3000, [2].ACC := 1167, [2].EN := 1, [2].TT := 1, [3].PRE := 3000, [3].ACC := 99, [3].EN := 1, [3].TT := 1, [4].PRE := 3000, [4].ACC := 98, [4].EN := 1, [4].TT := 1, [5].PRE := 3000, [5].ACC := 1221, [5].EN := 1, [5].TT := 1, [6].PRE := 3000, [6].ACC := 1013, [6].EN := 1, [6].TT := 1, [7].PRE := 3000, [7].ACC := 1220, [7].EN := 1, [7].TT := 1, [8].PRE := 3000, [8].ACC := 2381, [8].EN := 1, [8].TT := 1);
   Led_str_LenFix : Str_Len_Fix := (Len := 20);
   Led_strCMD : STRING[16] := ([0] := 'Z0$A1$01$01N$D0Test$00$00$00$00$00$00 2-1      R', [1] := 'Z0$A1$01$01N$D02026/04/29  10:28:16R', [2] := 'Z0$A1$01$01N$D0730000600  100.0 Kg R', [3] := 'Z0$A1$01$01N$D0BIN:41 3016E 5.00 t R', [4] := 'Z0$A1$01$01N$D0BIN:34 2410$00$00- 6.00tR', [5] := 'Z0$A1$01$01N$D02026/04/29  10:28:16R', [6] := 'Z0$A1$01$01N$D0S19-B8-2001B$00-99.0t R', [7] := 'Z0$A1$01$01N$D0S0-B139-3015$00$00- 3.0tR', [8] := 'Z0$A1$01$01N$D0BIN1 2001F$00-30.00t  R');
   Led_strOut : STRING[16] := ([0] := '$02Z0$A1$01$01N$D0Test$00$00$00$00$00$00 2-1      R?$03', [1] := '$02Z0$A1$01$01N$D02026/04/29  10:28:16R$02$03', [2] := '$02Z0$A1$01$01N$D0730000600  100.0 Kg R6$03', [3] := '$02Z0$A1$01$01N$D0BIN:41 3016E 5.00 t RS$03', [4] := '$02Z0$A1$01$01N$D0BIN:34 2410$00$00- 6.00tR9$03', [5] := '$02Z0$A1$01$01N$D02026/04/29  10:28:16R$02$03', [6] := '$02Z0$A1$01$01N$D0S19-B8-2001B$00-99.0t R$00$03', [7] := '$02Z0$A1$01$01N$D0S0-B139-3015$00$00- 3.0tRN$03', [8] := '$02Z0$A1$01$01N$D0BIN1 2001F$00-30.00t  Rb$03');
   TMP : DINT;
   UDP_Retry_T : TIMER := (PRE := 5000, ACC := 2019, EN := 1, TT := 1);
END_VAR

ROUTINE MainRoutine   (* ladder *)
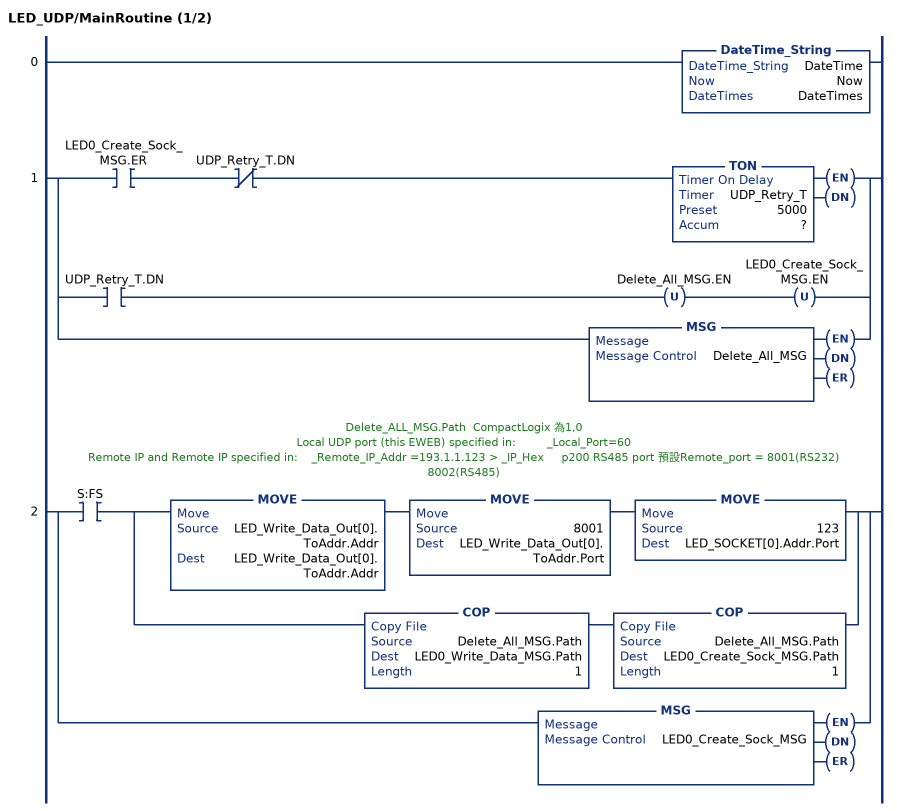
   0: DateTime_String(DateTime,Now,DateTimes);
   1: [XIC(LED0_Create_Sock_MSG.ER) XIO(UDP_Retry_T.DN) TON(UDP_Retry_T,?,?) ,XIC(UDP_Retry_T.DN) OTU(Delete_All_MSG.EN) OTU(LED0_Create_Sock_MSG.EN) ,MSG(Delete_All_MSG) ];
   // Delete_ALL_MSG.Path  CompactLogix 為1,0
   // Local UDP port (this EWEB) specified in:         _Local_Port=60
   // Remote IP and Remote IP specified in:    _Remote_IP_Addr =193.1.1.123 > _IP_Hex     p200 RS485 port 預設Remote_port = 8001(RS232) 8002(RS485)
   2: [XIC(S:FS) [MOVE(LED_Write_Data_Out[0].ToAddr.Addr,LED_Write_Data_Out[0].ToAddr.Addr) MOVE(8001,LED_Write_Data_Out[0].ToAddr.Port) MOVE(123,LED_SOCKET[0].Addr.Port) ,COP(Delete_All_MSG.Path,LED0_Write_Data_MSG.Path,1) COP(Delete_All_MSG.Path,LED0_Create_Sock_MSG.Path,1) ] ,MSG(LED0_Create_Sock_MSG) ];
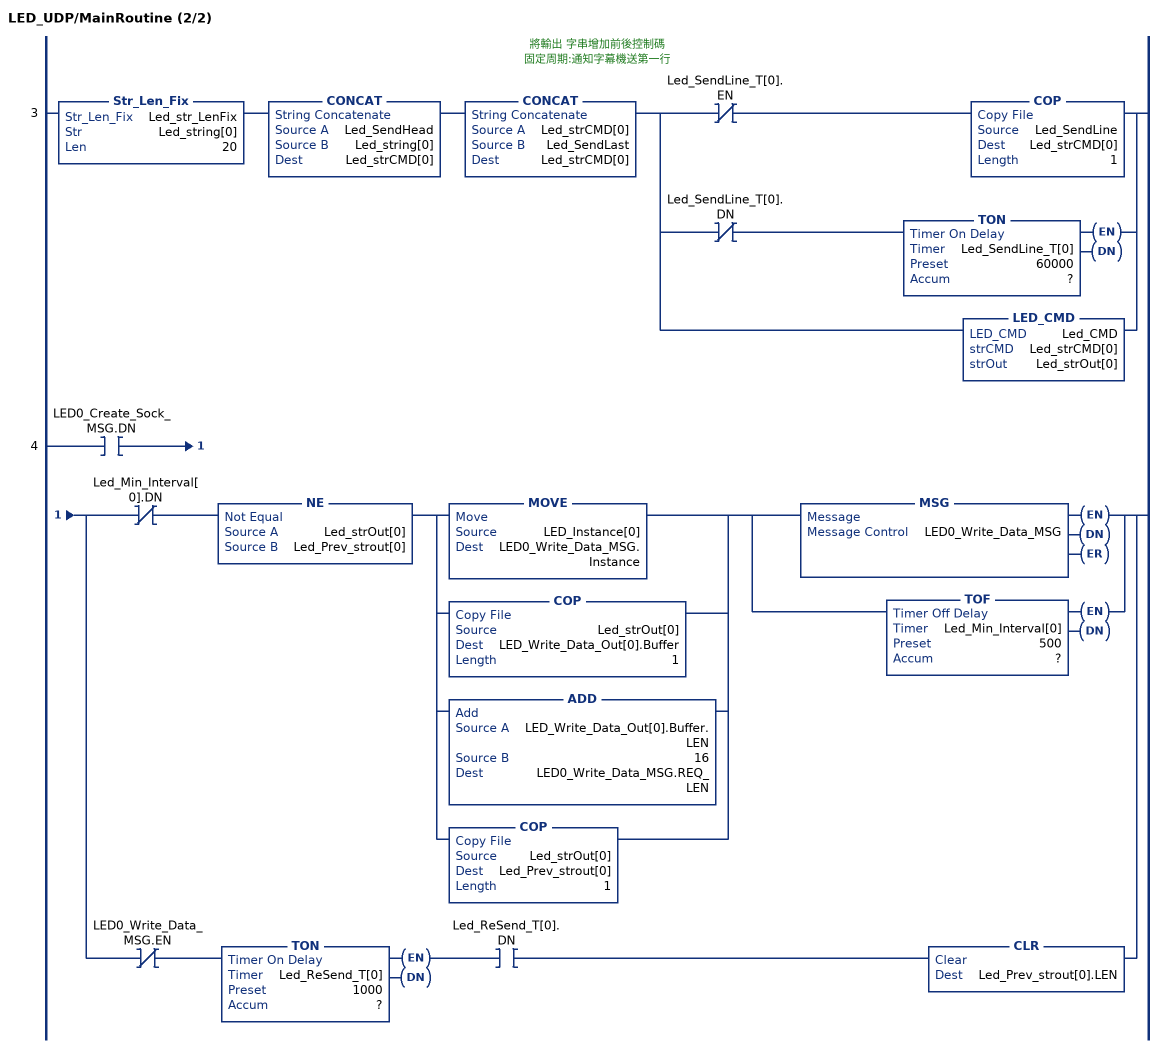
   // 將輸出 字串增加前後控制碼
   // 固定周期:通知字幕機送第一行
   3: Str_Len_Fix(Led_str_LenFix,Led_string[0],20)CONCAT(Led_SendHead,Led_string[0],Led_strCMD[0])CONCAT(Led_strCMD[0],Led_SendLast,Led_strCMD[0])[XIO(Led_SendLine_T[0].EN) COP(Led_SendLine,Led_strCMD[0],1) ,XIO(Led_SendLine_T[0].DN) TON(Led_SendLine_T[0],?,?) ,LED_CMD(Led_CMD,Led_strCMD[0],Led_strOut[0]) ];
   4: XIC(LED0_Create_Sock_MSG.DN)[XIO(Led_Min_Interval[0].DN) NE(Led_strOut[0],Led_Prev_strout[0]) [MOVE(LED_Instance[0],LED0_Write_Data_MSG.Instance) ,COP(Led_strOut[0],LED_Write_Data_Out[0].Buffer,1) ,ADD(LED_Write_Data_Out[0].Buffer.LEN,16,LED0_Write_Data_MSG.REQ_LEN) ,COP(Led_strOut[0],Led_Prev_strout[0],1) ] [MSG(LED0_Write_Data_MSG) ,TOF(Led_Min_Interval[0],?,?) ] ,XIO(LED0_Write_Data_MSG.EN) TON(Led_ReSend_T[0],?,?) XIC(Led_ReSend_T[0].DN) CLR(Led_Prev_strout[0].LEN) ];
END_ROUTINE
END_PROGRAM

PROGRAM MainProgram   (* main routine MainRoutine *)
VAR
   B126RPM : Speed_RPM := (RPM_Low := 60);
   B280_Delay : TIMER := (PRE := 500);
   ClearLog_T : TIMER := (PRE := 1000);
   Cow_SYS_B : System_Data;
   Cow_SYS_D : System_Data;
   Cow_SYS_E : System_Data := (MC := 1);
   Cow_SYS_F : System_Data;
   E120RPM : Speed_RPM := (RPM_Low := 60);
   Err_Reset_T : TIMER := (PRE := 1000);
   Logix_Type : DINT := 53;
   Ons : DINT;
   SYS_ON : BOOL := 1;
END_VAR
